Yaskawa INFORM job: PRINT3D17.JBI

/JOB
//NAME PRINT3D17
//POS
///NPOS 1138,0,0,0,0,0
///TOOL 9
///POSTYPE PULSE
///PULSE
C00000=35704,38341,-114719,81904,-122576,-81616,0
C00001=36579,38894,-113542,81280,-123389,-81453,0
C00002=42306,33068,-126081,74064,-124973,-85245,0
C00003=39937,31598,-129154,75978,-122913,-85572,0
C00004=34331,37524,-116454,82912,-121332,-81854,0
C00005=35234,38054,-115328,82245,-122145,-81700,0
C00006=34998,38355,-114678,82543,-122072,-81515,0
C00007=35467,38641,-114070,82205,-122503,-81430,0
C00008=35650,38409,-114572,81972,-122560,-81574,0
C00009=36212,38011,-115436,81348,-122827,-81855,0
C00010=36176,37331,-116893,81182,-122572,-82197,0
C00011=40262,33094,-125995,76081,-123713,-84903,0
C00012=40263,33039,-125991,76100,-123740,-84872,0
C00013=36399,37887,-115595,81173,-122955,-81890,0
C00014=41075,33073,-125931,75315,-124263,-84984,0
C00015=40068,32450,-127233,76121,-123383,-85125,0
C00016=35435,37299,-116842,81880,-122077,-82058,0
C00017=36321,37838,-115698,81229,-122883,-81904,0
C00018=35705,38292,-114715,81920,-122594,-81587,0
C00019=36579,38845,-113538,81297,-123409,-81425,0
C00020=42306,33013,-126077,74083,-125002,-85213,0
C00021=39937,31541,-129150,75996,-122940,-85539,0
C00022=34332,37475,-116451,82927,-121351,-81824,0
C00023=35234,38005,-115325,82261,-122164,-81671,0
C00024=34998,38306,-114675,82559,-122092,-81485,0
C00025=35467,38592,-114066,82221,-122522,-81401,0
C00026=35650,38360,-114568,81989,-122578,-81545,0
C00027=36212,37961,-115433,81364,-122847,-81826,0
C00028=36177,37281,-116890,81199,-122593,-82168,0
C00029=40263,33039,-125991,76100,-123740,-84872,0
C00030=40263,32984,-125988,76119,-123766,-84840,0
C00031=36400,37838,-115591,81189,-122975,-81861,0
C00032=41075,33018,-125927,75334,-124289,-84952,0
C00033=40068,32394,-127230,76140,-123410,-85093,0
C00034=35436,37249,-116838,81896,-122097,-82028,0
C00035=36322,37789,-115695,81246,-122903,-81874,0
C00036=35705,38243,-114712,81937,-122614,-81558,0
C00037=36579,38797,-113534,81314,-123427,-81396,0
C00038=42306,32958,-126074,74103,-125029,-85181,0
C00039=39938,31484,-129146,76015,-122968,-85507,0
C00040=34332,37425,-116447,82943,-121369,-81794,0
C00041=35235,37956,-115321,82277,-122183,-81642,0
C00042=34998,38257,-114671,82575,-122110,-81456,0
C00043=35467,38544,-114062,82237,-122540,-81372,0
C00044=35651,38311,-114564,82005,-122597,-81516,0
C00045=36213,37912,-115428,81381,-122867,-81797,0
C00046=36177,37232,-116886,81215,-122613,-82137,0
C00047=40263,32984,-125988,76119,-123766,-84840,0
C00048=40264,32929,-125983,76137,-123793,-84808,0
C00049=36400,37788,-115587,81206,-122994,-81831,0
C00050=41076,32964,-125923,75353,-124317,-84920,0
C00051=40069,32339,-127226,76159,-123437,-85061,0
C00052=35436,37199,-116833,81912,-122116,-81998,0
C00053=36322,37739,-115690,81263,-122923,-81845,0
C00054=35705,38194,-114708,81953,-122633,-81529,0
C00055=36580,38748,-113531,81331,-123447,-81367,0
C00056=42307,32903,-126069,74123,-125058,-85150,0
C00057=39938,31428,-129142,76033,-122995,-85474,0
C00058=34332,37375,-116443,82958,-121388,-81765,0
C00059=35235,37907,-115318,82293,-122201,-81612,0
C00060=34999,38208,-114667,82591,-122129,-81427,0
C00061=35468,38495,-114059,82254,-122560,-81343,0
C00062=35651,38262,-114561,82021,-122616,-81487,0
C00063=36213,37863,-115425,81398,-122886,-81767,0
C00064=36178,37182,-116883,81232,-122633,-82108,0
C00065=40264,32929,-125983,76137,-123793,-84808,0
C00066=40264,32874,-125980,76156,-123820,-84777,0
C00067=36400,37739,-115583,81223,-123015,-81802,0
C00068=41076,32909,-125919,75372,-124344,-84888,0
C00069=40069,32283,-127222,76177,-123463,-85029,0
C00070=35436,37150,-116830,81928,-122135,-81968,0
C00071=36322,37690,-115687,81279,-122942,-81816,0
C00072=35706,38145,-114704,81969,-122652,-81500,0
C00073=36580,38700,-113527,81348,-123466,-81338,0
C00074=42307,32849,-126066,74142,-125087,-85119,0
C00075=39938,31371,-129138,76052,-123023,-85442,0
C00076=34333,37326,-116439,82974,-121406,-81735,0
C00077=35235,37857,-115313,82310,-122221,-81583,0
C00078=34999,38160,-114663,82607,-122147,-81397,0
C00079=35468,38447,-114055,82270,-122578,-81314,0
C00080=35651,38214,-114557,82038,-122634,-81457,0
C00081=36213,37814,-115421,81414,-122906,-81738,0
C00082=36178,37132,-116878,81249,-122653,-82078,0
C00083=40264,32874,-125980,76156,-123820,-84777,0
C00084=40264,32820,-125975,76175,-123847,-84745,0
C00085=36401,37690,-115580,81240,-123034,-81772,0
C00086=41077,32854,-125915,75391,-124371,-84857,0
C00087=40070,32228,-127218,76196,-123491,-84997,0
C00088=35437,37100,-116827,81945,-122154,-81939,0
C00089=36323,37641,-115683,81296,-122962,-81786,0
C00090=35706,38096,-114700,81986,-122671,-81470,0
C00091=36580,38652,-113523,81365,-123486,-81309,0
C00092=42308,32794,-126061,74162,-125115,-85087,0
C00093=39939,31314,-129134,76070,-123050,-85409,0
C00094=34333,37276,-116436,82989,-121424,-81706,0
C00095=35236,37808,-115310,82326,-122239,-81554,0
C00096=34999,38111,-114660,82623,-122166,-81368,0
C00097=35468,38398,-114051,82286,-122597,-81284,0
C00098=35652,38165,-114553,82054,-122654,-81428,0
C00099=36214,37764,-115417,81431,-122925,-81709,0
C00100=36178,37082,-116875,81265,-122672,-82049,0
C00101=40264,32820,-125975,76175,-123847,-84745,0
C00102=40265,32765,-125972,76194,-123873,-84713,0
C00103=36401,37640,-115575,81256,-123054,-81743,0
C00104=41077,32800,-125911,75411,-124398,-84825,0
C00105=40070,32173,-127214,76215,-123517,-84965,0
C00106=35437,37050,-116822,81961,-122174,-81909,0
C00107=36323,37592,-115679,81313,-122981,-81757,0
C00108=35706,38048,-114696,82002,-122690,-81441,0
C00109=36580,38604,-113519,81382,-123505,-81280,0
C00110=42308,32739,-126058,74182,-125143,-85055,0
C00111=39939,31258,-129129,76089,-123078,-85376,0
C00112=34333,37226,-116431,83005,-121444,-81676,0
C00113=35236,37759,-115306,82342,-122259,-81524,0
C00114=35000,38062,-114656,82639,-122184,-81339,0
C00115=35469,38350,-114047,82303,-122615,-81255,0
C00116=35652,38116,-114549,82071,-122672,-81399,0
C00117=36214,37715,-115413,81448,-122946,-81679,0
C00118=36179,37032,-116870,81282,-122693,-82018,0
C00119=40265,32765,-125972,76194,-123873,-84713,0
C00120=40265,32711,-125967,76213,-123900,-84682,0
C00121=36401,37591,-115572,81273,-123073,-81713,0
C00122=41077,32745,-125906,75430,-124426,-84794,0
C00123=40070,32117,-127209,76233,-123545,-84933,0
C00124=35437,37000,-116819,81977,-122193,-81879,0
C00125=36323,37542,-115675,81330,-123002,-81727,0
C00126=35707,37999,-114692,82019,-122709,-81411,0
C00127=36581,38555,-113515,81399,-123525,-81251,0
C00128=42309,32685,-126053,74202,-125172,-85024,0
C00129=39940,31201,-129125,76108,-123106,-85344,0
C00130=34333,37177,-116427,83021,-121462,-81646,0
C00131=35236,37710,-115302,82358,-122277,-81494,0
C00132=35000,38013,-114651,82655,-122202,-81310,0
C00133=35469,38301,-114043,82319,-122634,-81226,0
C00134=35652,38067,-114545,82087,-122692,-81370,0
C00135=36214,37666,-115409,81465,-122965,-81649,0
C00136=36179,36982,-116867,81299,-122713,-81989,0
C00137=40265,32711,-125967,76213,-123900,-84682,0
C00138=40266,32656,-125962,76232,-123926,-84650,0
C00139=36402,37542,-115567,81290,-123094,-81684,0
C00140=41078,32691,-125903,75449,-124454,-84762,0
C00141=40071,32062,-127205,76252,-123571,-84901,0
C00142=35438,36951,-116814,81994,-122213,-81849,0
C00143=36324,37493,-115671,81347,-123022,-81697,0
C00144=35707,37950,-114688,82035,-122728,-81382,0
C00145=36581,38507,-113511,81416,-123545,-81222,0
C00146=42309,32630,-126049,74222,-125200,-84993,0
C00147=39940,31145,-129120,76126,-123133,-85311,0
C00148=34334,37127,-116423,83036,-121481,-81616,0
C00149=35237,37661,-115297,82374,-122295,-81465,0
C00150=35000,37965,-114647,82671,-122221,-81280,0
C00151=35469,38253,-114039,82335,-122653,-81197,0
C00152=35653,38019,-114541,82104,-122710,-81340,0
C00153=36215,37617,-115405,81481,-122985,-81620,0
C00154=36179,36933,-116862,81315,-122733,-81959,0
C00155=40266,32656,-125962,76232,-123926,-84650,0
C00156=40266,32601,-125958,76250,-123953,-84618,0
C00157=36402,37493,-115563,81307,-123114,-81655,0
C00158=41078,32636,-125898,75469,-124480,-84731,0
C00159=40071,32007,-127201,76271,-123597,-84869,0
C00160=35438,36901,-116809,82010,-122232,-81819,0
C00161=36324,37444,-115666,81363,-123041,-81668,0
C00162=35707,37901,-114684,82052,-122747,-81353,0
C00163=36581,38459,-113507,81433,-123563,-81193,0
C00164=42309,32575,-126044,74242,-125229,-84961,0
C00165=39940,31088,-129117,76145,-123161,-85278,0
C00166=34334,37078,-116419,83052,-121499,-81587,0
C00167=35237,37612,-115294,82391,-122315,-81435,0
C00168=35001,37916,-114643,82687,-122239,-81251,0
C00169=35470,38204,-114035,82352,-122671,-81168,0
C00170=35653,37970,-114537,82120,-122730,-81311,0
C00171=36215,37568,-115400,81498,-123004,-81591,0
C00172=36179,36883,-116859,81332,-122753,-81929,0
C00173=40266,32601,-125958,76250,-123953,-84618,0
C00174=40266,32547,-125953,76269,-123979,-84586,0
C00175=36402,37444,-115559,81324,-123133,-81625,0
C00176=41079,32582,-125893,75488,-124508,-84699,0
C00177=40072,31951,-127197,76290,-123625,-84836,0
C00178=35438,36851,-116805,82026,-122252,-81789,0
C00179=36324,37395,-115663,81380,-123061,-81638,0
C00180=35707,37853,-114679,82068,-122765,-81324,0
C00181=36582,38411,-113502,81450,-123582,-81163,0
C00182=42310,32521,-126039,74262,-125257,-84930,0
C00183=39941,31032,-129112,76164,-123188,-85245,0
C00184=34335,37028,-116414,83068,-121517,-81556,0
C00185=35237,37563,-115289,82407,-122333,-81406,0
C00186=35001,37867,-114639,82704,-122258,-81222,0
C00187=35470,38156,-114030,82368,-122690,-81139,0
C00188=35653,37921,-114532,82137,-122748,-81281,0
C00189=36215,37519,-115396,81515,-123024,-81561,0
C00190=36180,36833,-116854,81349,-122772,-81899,0
C00191=40266,32547,-125953,76269,-123979,-84586,0
C00192=40267,32493,-125949,76288,-124005,-84554,0
C00193=36403,37395,-115554,81341,-123153,-81595,0
C00194=41079,32527,-125889,75508,-124535,-84667,0
C00195=40072,31896,-127192,76309,-123651,-84804,0
C00196=35439,36802,-116801,82043,-122271,-81760,0
C00197=36325,37346,-115658,81397,-123080,-81609,0
C00198=35708,37804,-114675,82085,-122785,-81294,0
C00199=36582,38363,-113498,81467,-123602,-81134,0
C00200=42310,32466,-126035,74282,-125286,-84898,0
C00201=39941,30975,-129108,76183,-123216,-85213,0
C00202=34335,36979,-116411,83084,-121536,-81527,0
C00203=35237,37515,-115284,82423,-122353,-81376,0
C00204=35001,37819,-114634,82720,-122276,-81192,0
C00205=35470,38108,-114026,82385,-122708,-81109,0
C00206=35654,37873,-114528,82153,-122768,-81252,0
C00207=36216,37470,-115392,81532,-123044,-81532,0
C00208=36180,36784,-116850,81366,-122793,-81869,0
C00209=40267,32493,-125949,76288,-124005,-84554,0
C00210=40267,32438,-125944,76307,-124033,-84522,0
C00211=36403,37346,-115550,81358,-123172,-81566,0
C00212=41079,32473,-125884,75527,-124563,-84635,0
C00213=40072,31841,-127187,76328,-123679,-84772,0
C00214=35439,36752,-116797,82059,-122291,-81729,0
C00215=36325,37297,-115653,81414,-123101,-81579,0
C00216=35708,37756,-114671,82102,-122803,-81265,0
C00217=36583,38315,-113493,81484,-123622,-81105,0
C00218=42311,32412,-126030,74302,-125314,-84866,0
C00219=39942,30919,-129102,76202,-123243,-85180,0
C00220=34335,36930,-116406,83099,-121554,-81497,0
C00221=35238,37466,-115280,82440,-122371,-81346,0
C00222=35002,37770,-114630,82736,-122294,-81162,0
C00223=35471,38059,-114022,82401,-122728,-81080,0
C00224=35654,37825,-114523,82170,-122786,-81223,0
C00225=36216,37421,-115388,81549,-123063,-81502,0
C00226=36180,36734,-116845,81383,-122813,-81840,0
C00227=40267,32438,-125944,76307,-124033,-84522,0
C00228=40268,32384,-125939,76327,-124059,-84490,0
C00229=36403,37297,-115545,81375,-123193,-81536,0
C00230=41080,32419,-125880,75547,-124589,-84603,0
C00231=40073,31786,-127182,76347,-123705,-84739,0
C00232=35439,36703,-116792,82076,-122309,-81700,0
C00233=36325,37248,-115649,81431,-123121,-81550,0
C00234=35709,37707,-114666,82118,-122823,-81235,0
C00235=36583,38267,-113489,81502,-123641,-81076,0
C00236=42311,32358,-126026,74322,-125342,-84834,0
C00237=39942,30863,-129097,76221,-123271,-85147,0
C00238=34335,36880,-116401,83115,-121573,-81467,0
C00239=35238,37417,-115275,82456,-122390,-81317,0
C00240=35002,37722,-114625,82752,-122313,-81133,0
C00241=35471,38011,-114017,82418,-122746,-81050,0
C00242=35654,37776,-114519,82187,-122806,-81193,0
C00243=36216,37373,-115383,81566,-123083,-81472,0
C00244=36181,36685,-116840,81400,-122833,-81809,0
C00245=40268,32384,-125939,76327,-124059,-84490,0
C00246=40268,32330,-125935,76346,-124086,-84458,0
C00247=36404,37248,-115541,81392,-123212,-81507,0
C00248=41080,32364,-125875,75566,-124617,-84572,0
C00249=40073,31731,-127177,76366,-123733,-84707,0
C00250=35440,36653,-116788,82092,-122329,-81670,0
C00251=36326,37199,-115644,81448,-123140,-81520,0
C00252=35709,37659,-114661,82135,-122841,-81206,0
C00253=36583,38219,-113484,81519,-123659,-81046,0
C00254=42312,32303,-126021,74342,-125371,-84802,0
C00255=39943,30806,-129093,76240,-123299,-85114,0
C00256=34336,36831,-116397,83131,-121591,-81437,0
C00257=35239,37368,-115271,82472,-122409,-81287,0
C00258=35002,37673,-114621,82769,-122331,-81103,0
C00259=35471,37963,-114012,82434,-122764,-81021,0
C00260=35655,37728,-114514,82203,-122824,-81164,0
C00261=36217,37324,-115379,81583,-123102,-81443,0
C00262=36181,36635,-116836,81417,-122853,-81780,0
C00263=40268,32330,-125935,76346,-124086,-84458,0
C00264=40268,32275,-125930,76365,-124112,-84426,0
C00265=36404,37200,-115536,81410,-123232,-81476,0
C00266=41081,32310,-125869,75586,-124644,-84540,0
C00267=40074,31676,-127172,76385,-123759,-84675,0
C00268=35440,36604,-116783,82109,-122348,-81639,0
C00269=36326,37150,-115640,81465,-123160,-81490,0
C00270=35709,37610,-114657,82152,-122861,-81176,0
C00271=36583,38171,-113480,81536,-123679,-81017,0
C00272=42312,32249,-126016,74362,-125399,-84771,0
C00273=39943,30750,-129087,76259,-123326,-85081,0
C00274=34336,36782,-116392,83147,-121609,-81407,0
C00275=35239,37319,-115266,82489,-122428,-81258,0
C00276=35003,37625,-114616,82785,-122349,-81074,0
C00277=35472,37915,-114008,82451,-122783,-80992,0
C00278=35655,37679,-114510,82220,-122844,-81135,0
C00279=36217,37275,-115374,81600,-123122,-81413,0
C00280=36182,36586,-116831,81434,-122872,-81750,0
C00281=40268,32275,-125930,76365,-124112,-84426,0
C00282=40269,32221,-125924,76384,-124139,-84395,0
C00283=36404,37151,-115532,81427,-123252,-81447,0
C00284=41081,32256,-125865,75605,-124672,-84508,0
C00285=40074,31621,-127167,76404,-123786,-84642,0
C00286=35440,36555,-116777,82125,-122368,-81610,0
C00287=36326,37101,-115635,81483,-123179,-81461,0
C00288=35710,37562,-114652,82168,-122880,-81147,0
C00289=36584,38123,-113475,81553,-123699,-80988,0
C00290=42312,32195,-126011,74383,-125428,-84739,0
C00291=39943,30694,-129082,76278,-123354,-85048,0
C00292=34336,36733,-116386,83163,-121628,-81377,0
C00293=35239,37271,-115261,82505,-122446,-81228,0
C00294=35003,37576,-114611,82801,-122369,-81045,0
C00295=35472,37867,-114003,82467,-122802,-80962,0
C00296=35655,37631,-114505,82237,-122862,-81105,0
C00297=36217,37226,-115368,81617,-123141,-81384,0
C00298=36182,36536,-116827,81451,-122893,-81720,0
C00299=40269,32221,-125924,76384,-124139,-84395,0
C00300=40269,32167,-125920,76404,-124165,-84363,0
C00301=36405,37102,-115526,81444,-123271,-81417,0
C00302=41082,32202,-125859,75625,-124698,-84476,0
C00303=40074,31566,-127162,76423,-123813,-84610,0
C00304=35441,36505,-116773,82142,-122387,-81580,0
C00305=36327,37053,-115629,81500,-123200,-81431,0
C00306=35710,37513,-114647,82185,-122899,-81117,0
C00307=36584,38075,-113470,81571,-123718,-80959,0
C00308=42313,32140,-126006,74403,-125456,-84707,0
C00309=39944,30638,-129078,76297,-123381,-85015,0
C00310=34337,36683,-116382,83179,-121646,-81347,0
C00311=35239,37222,-115257,82522,-122466,-81198,0
C00312=35003,37528,-114606,82818,-122387,-81015,0
C00313=35472,37819,-113998,82484,-122821,-80933,0
C00314=35656,37583,-114500,82253,-122882,-81075,0
C00315=36218,37178,-115364,81634,-123161,-81353,0
C00316=36182,36487,-116821,81468,-122913,-81690,0
C00317=40269,32167,-125920,76404,-124165,-84363,0
C00318=40270,32113,-125914,76423,-124192,-84331,0
C00319=36405,37053,-115521,81461,-123292,-81388,0
C00320=41082,32148,-125854,75645,-124726,-84444,0
C00321=40075,31511,-127156,76443,-123840,-84577,0
C00322=35441,36456,-116768,82159,-122407,-81550,0
C00323=36327,37004,-115625,81517,-123219,-81401,0
C00324=35710,37465,-114642,82202,-122918,-81088,0
C00325=36584,38027,-113465,81588,-123738,-80930,0
C00326=42313,32086,-126000,74423,-125484,-84675,0
C00327=39944,30582,-129072,76316,-123409,-84982,0
C00328=34337,36634,-116377,83195,-121665,-81317,0
C00329=35240,37174,-115251,82538,-122484,-81168,0
C00330=35004,37480,-114601,82834,-122406,-80985,0
C00331=35472,37771,-113993,82501,-122839,-80904,0
C00332=35656,37534,-114495,82270,-122900,-81046,0
C00333=36218,37129,-115359,81651,-123180,-81324,0
C00334=36183,36438,-116816,81485,-122933,-81660,0
C00335=40270,32113,-125914,76423,-124192,-84331,0
C00336=40270,32059,-125910,76442,-124218,-84298,0
C00337=36405,37005,-115517,81478,-123311,-81357,0
C00338=41082,32094,-125849,75665,-124753,-84412,0
C00339=40075,31456,-127152,76462,-123867,-84545,0
C00340=35441,36407,-116762,82175,-122426,-81519,0
C00341=36327,36955,-115620,81534,-123239,-81371,0
C00342=35710,37417,-114637,82219,-122937,-81058,0
C00343=36585,37980,-113460,81605,-123757,-80900,0
C00344=42314,32032,-125996,74444,-125513,-84643,0
C00345=39945,30526,-129066,76335,-123437,-84949,0
C00346=34337,36585,-116372,83211,-121683,-81287,0
C00347=35240,37125,-115247,82555,-122502,-81139,0
C00348=35004,37432,-114596,82850,-122424,-80956,0
C00349=35473,37723,-113988,82517,-122857,-80874,0
C00350=35656,37486,-114490,82287,-122918,-81016,0
C00351=36218,37080,-115353,81668,-123200,-81294,0
C00352=36183,36388,-116812,81502,-122953,-81630,0
C00353=40270,32059,-125910,76442,-124218,-84298,0
C00354=40271,32005,-125904,76462,-124244,-84266,0
C00355=36406,36956,-115511,81496,-123331,-81328,0
C00356=41083,32040,-125844,75684,-124780,-84380,0
C00357=40076,31402,-127146,76481,-123894,-84513,0
C00358=35442,36358,-116758,82192,-122446,-81489,0
C00359=36328,36906,-115614,81551,-123258,-81341,0
C00360=35711,37369,-114632,82236,-122956,-81028,0
C00361=36585,37932,-113455,81623,-123776,-80871,0
C00362=42314,31978,-125990,74464,-125542,-84612,0
C00363=39945,30470,-129061,76354,-123464,-84916,0
C00364=34338,36536,-116367,83227,-121701,-81257,0
C00365=35240,37077,-115241,82572,-122522,-81109,0
C00366=35004,37383,-114591,82867,-122443,-80926,0
C00367=35473,37675,-113983,82534,-122876,-80844,0
C00368=35657,37438,-114485,82304,-122938,-80987,0
C00369=36219,37032,-115349,81685,-123219,-81265,0
C00370=36183,36339,-116806,81519,-122972,-81599,0
C00371=40271,32005,-125904,76462,-124244,-84266,0
C00372=40271,31951,-125898,76481,-124272,-84234,0
C00373=36406,36908,-115506,81513,-123350,-81298,0
C00374=41083,31986,-125838,75704,-124807,-84348,0
C00375=40076,31347,-127140,76501,-123920,-84480,0
C00376=35442,36308,-116752,82209,-122464,-81459,0
C00377=36328,36858,-115610,81569,-123278,-81312,0
C00378=35711,37320,-114627,82253,-122975,-80999,0
C00379=36585,37884,-113450,81640,-123795,-80842,0
C00380=42315,31924,-125984,74485,-125569,-84580,0
C00381=39945,30414,-129056,76374,-123492,-84883,0
C00382=34338,36487,-116361,83243,-121720,-81227,0
C00383=35241,37028,-115236,82588,-122540,-81080,0
C00384=35005,37335,-114586,82883,-122461,-80896,0
C00385=35474,37627,-113978,82551,-122895,-80815,0
C00386=35657,37390,-114480,82321,-122956,-80957,0
C00387=36219,36983,-115343,81703,-123239,-81234,0
C00388=36184,36290,-116801,81536,-122993,-81569,0
C00389=40271,31951,-125898,76481,-124272,-84234,0
C00390=40271,31897,-125892,76501,-124298,-84202,0
C00391=36406,36859,-115500,81530,-123371,-81268,0
C00392=41084,31932,-125833,75724,-124835,-84316,0
C00393=40076,31292,-127135,76520,-123948,-84447,0
C00394=35442,36259,-116747,82226,-122484,-81429,0
C00395=36328,36809,-115604,81586,-123297,-81281,0
C00396=35711,37272,-114621,82270,-122994,-80969,0
C00397=36586,37837,-113444,81658,-123815,-80812,0
C00398=42315,31870,-125978,74505,-125598,-84548,0
C00399=39946,30358,-129050,76393,-123519,-84849,0
C00400=34338,36438,-116357,83259,-121738,-81197,0
C00401=35241,36980,-115230,82605,-122560,-81049,0
C00402=35005,37287,-114581,82900,-122479,-80867,0
C00403=35474,37579,-113972,82568,-122914,-80785,0
C00404=35657,37342,-114474,82338,-122976,-80927,0
C00405=36219,36935,-115338,81720,-123258,-81205,0
C00406=36184,36241,-116796,81554,-123013,-81539,0
C00407=40271,31897,-125892,76501,-124298,-84202,0
C00408=40272,31843,-125888,76520,-124325,-84170,0
C00409=36407,36811,-115495,81548,-123391,-81238,0
C00410=41084,31878,-125827,75744,-124863,-84284,0
C00411=40077,31238,-127129,76539,-123974,-84415,0
C00412=35443,36210,-116742,82242,-122503,-81399,0
C00413=36329,36761,-115598,81603,-123318,-81252,0
C00414=35712,37224,-114616,82287,-123013,-80939,0
C00415=36586,37789,-113439,81675,-123834,-80783,0
C00416=42315,31816,-125973,74526,-125627,-84516,0
C00417=39946,30302,-129044,76412,-123547,-84816,0
C00418=34339,36389,-116351,83275,-121756,-81167,0
C00419=35241,36931,-115226,82622,-122578,-81020,0
C00420=35005,37239,-114575,82916,-122498,-80837,0
C00421=35474,37531,-113967,82585,-122932,-80756,0
C00422=35658,37294,-114469,82355,-122994,-80898,0
C00423=36220,36887,-115333,81737,-123278,-81175,0
C00424=36184,36192,-116790,81571,-123032,-81509,0
C00425=40272,31843,-125888,76520,-124325,-84170,0
C00426=40272,31789,-125882,76540,-124351,-84138,0
C00427=36407,36762,-115490,81565,-123410,-81208,0
C00428=41084,31824,-125821,75764,-124889,-84252,0
C00429=40077,31183,-127123,76559,-124001,-84382,0
C00430=35443,36161,-116736,82259,-122523,-81368,0
C00431=36329,36712,-115592,81621,-123338,-81222,0
C00432=35712,37176,-114611,82304,-123032,-80909,0
C00433=36586,37742,-113434,81693,-123854,-80753,0
C00434=42316,31762,-125968,74546,-125654,-84484,0
C00435=39947,30246,-129039,76432,-123574,-84783,0
C00436=34339,36341,-116345,83292,-121775,-81136,0
C00437=35242,36883,-115220,82638,-122597,-80990,0
C00438=35006,37191,-114570,82933,-122516,-80807,0
C00439=35474,37483,-113962,82601,-122950,-80726,0
C00440=35658,37246,-114463,82371,-123014,-80868,0
C00441=36220,36838,-115327,81754,-123297,-81145,0
C00442=36185,36143,-116784,81588,-123053,-81479,0
C00443=40272,31789,-125882,76540,-124351,-84138,0
C00444=40273,31735,-125876,76559,-124378,-84106,0
C00445=36407,36714,-115484,81583,-123430,-81179,0
C00446=41085,31770,-125815,75784,-124917,-84219,0
C00447=40078,31128,-127117,76578,-124028,-84350,0
C00448=35443,36112,-116730,82276,-122543,-81338,0
C00449=36329,36664,-115588,81638,-123357,-81192,0
C00450=35713,37128,-114605,82321,-123050,-80880,0
C00451=36587,37694,-113428,81710,-123872,-80724,0
C00452=42316,31708,-125961,74567,-125683,-84452,0
C00453=39947,30191,-129033,76451,-123602,-84750,0
C00454=34339,36292,-116339,83308,-121793,-81106,0
C00455=35242,36835,-115214,82655,-122616,-80960,0
C00456=35006,37143,-114564,82949,-122534,-80777,0
C00457=35475,37436,-113956,82618,-122969,-80697,0
C00458=35658,37198,-114458,82388,-123032,-80838,0
C00459=36220,36790,-115322,81772,-123317,-81115,0
C00460=36185,36094,-116779,81605,-123072,-81449,0
C00461=40273,31735,-125876,76559,-124378,-84106,0
C00462=40273,31682,-125869,76579,-124404,-84073,0
C00463=36408,36665,-115479,81600,-123449,-81149,0
C00464=41085,31717,-125810,75804,-124944,-84187,0
C00465=40078,31074,-127112,76598,-124055,-84317,0
C00466=35444,36063,-116724,82293,-122562,-81308,0
C00467=36330,36615,-115582,81655,-123377,-81162,0
C00468=35713,37080,-114599,82338,-123070,-80850,0
C00469=36587,37647,-113422,81728,-123892,-80694,0
C00470=42317,31655,-125955,74588,-125712,-84420,0
C00471=39948,30135,-129026,76471,-123630,-84717,0
C00472=34340,36243,-116334,83324,-121812,-81076,0
C00473=35242,36786,-115209,82672,-122634,-80930,0
C00474=35006,37095,-114559,82966,-122553,-80748,0
C00475=35475,37388,-113950,82635,-122988,-80667,0
C00476=35659,37150,-114452,82405,-123052,-80809,0
C00477=36221,36742,-115317,81789,-123337,-81085,0
C00478=36185,36045,-116774,81623,-123093,-81418,0
C00479=40273,31682,-125869,76579,-124404,-84073,0
C00480=40273,31628,-125864,76599,-124431,-84041,0
C00481=36408,36617,-115473,81618,-123469,-81118,0
C00482=41086,31663,-125804,75824,-124971,-84155,0
C00483=40079,31020,-127106,76617,-124082,-84285,0
C00484=35444,36014,-116719,82310,-122582,-81278,0
C00485=36330,36567,-115576,81673,-123396,-81132,0
C00486=35713,37032,-114594,82355,-123088,-80820,0
C00487=36587,37599,-113417,81746,-123911,-80665,0
C00488=42317,31601,-125950,74608,-125741,-84388,0
C00489=39948,30079,-129020,76490,-123657,-84684,0
C00490=34340,36194,-116328,83340,-121830,-81046,0
C00491=35243,36738,-115203,82689,-122653,-80900,0
C00492=35006,37047,-114553,82983,-122571,-80718,0
C00493=35475,37340,-113945,82652,-123007,-80637,0
C00494=35659,37102,-114447,82423,-123070,-80779,0
C00495=36221,36693,-115311,81807,-123356,-81055,0
C00496=36186,35996,-116768,81640,-123112,-81388,0
C00497=40273,31628,-125864,76599,-124431,-84041,0
C00498=40274,31574,-125858,76618,-124457,-84009,0
C00499=36408,36569,-115467,81635,-123489,-81089,0
C00500=41086,31609,-125798,75844,-124998,-84123,0
C00501=40079,30965,-127100,76637,-124109,-84252,0
C00502=35444,35965,-116713,82327,-122600,-81248,0
C00503=36330,36519,-115571,81690,-123416,-81102,0
C00504=35713,36984,-114588,82372,-123108,-80791,0
C00505=36588,37552,-113411,81763,-123931,-80635,0
C00506=42318,31547,-125944,74629,-125768,-84356,0
C00507=39948,30024,-129015,76510,-123684,-84650,0
C00508=35603,34554,-119651,81803,-122284,-81944,0
C00509=35599,34552,-119656,81806,-122280,-81945,0
C00510=35261,34964,-118796,82221,-122166,-81703,0
C00511=35265,34966,-118792,82218,-122168,-81703,0
C00512=34340,36146,-116322,83357,-121848,-81016,0
C00513=35243,36690,-115197,82705,-122672,-80870,0
C00514=35007,36999,-114547,82999,-122590,-80688,0
C00515=35476,37293,-113939,82669,-123025,-80608,0
C00516=35659,37054,-114441,82440,-123088,-80749,0
C00517=36221,36645,-115305,81824,-123376,-81026,0
C00518=36186,35947,-116762,81657,-123132,-81358,0
C00519=40274,31574,-125858,76618,-124457,-84009,0
C00520=40274,31521,-125852,76638,-124483,-83976,0
C00521=36409,36520,-115461,81653,-123509,-81059,0
C00522=41086,31556,-125791,75865,-125026,-84091,0
C00523=40079,30911,-127093,76657,-124135,-84219,0
C00524=35445,35917,-116707,82344,-122619,-81217,0
C00525=36331,36470,-115565,81708,-123437,-81072,0
C00526=35714,36937,-114582,82389,-123126,-80760,0
C00527=36588,37505,-113405,81781,-123950,-80605,0
C00528=42318,31493,-125938,74650,-125797,-84323,0
C00529=39949,29968,-129008,76530,-123711,-84617,0
C00530=35603,34504,-119645,81820,-122303,-81913,0
C00531=35585,34493,-119667,81834,-122287,-81916,0
C00532=35247,34905,-118808,82249,-122172,-81675,0
C00533=35265,34916,-118786,82235,-122189,-81672,0
C00534=34341,36097,-116316,83373,-121867,-80985,0
C00535=35243,36642,-115191,82722,-122691,-80840,0
C00536=35007,36951,-114541,83016,-122608,-80658,0
C00537=35476,37245,-113933,82686,-123044,-80578,0
C00538=35659,37007,-114435,82457,-123108,-80719,0
C00539=36222,36597,-115298,81841,-123395,-80995,0
C00540=36186,35898,-116755,81675,-123153,-81327,0
C00541=40274,31521,-125852,76638,-124483,-83976,0
C00542=40275,31467,-125845,76658,-124510,-83944,0
C00543=36409,36472,-115455,81670,-123528,-81028,0
C00544=41087,31502,-125785,75885,-125052,-84059,0
C00545=40080,30856,-127087,76676,-124163,-84186,0
C00546=35445,35868,-116701,82361,-122639,-81187,0
C00547=36331,36422,-115558,81726,-123456,-81042,0
C00548=35714,36889,-114576,82406,-123146,-80731,0
C00549=36588,37457,-113399,81799,-123969,-80576,0
C00550=42318,31440,-125931,74671,-125826,-84291,0
C00551=39949,29913,-129002,76549,-123739,-84584,0
C00552=35604,34453,-119640,81837,-122324,-81882,0
C00553=35571,34434,-119679,81862,-122295,-81887,0
C00554=35233,34847,-118819,82276,-122179,-81646,0
C00555=35266,34866,-118779,82252,-122208,-81641,0
C00556=34341,36048,-116311,83389,-121885,-80955,0
C00557=35244,36594,-115186,82739,-122709,-80810,0
C00558=35007,36904,-114535,83033,-122626,-80628,0
C00559=35476,37198,-113927,82703,-123062,-80548,0
C00560=35660,36959,-114429,82474,-123126,-80690,0
C00561=36222,36549,-115292,81859,-123415,-80965,0
C00562=36187,35849,-116750,81692,-123172,-81297,0
C00563=40275,31467,-125845,76658,-124510,-83944,0
C00564=40275,31413,-125839,76678,-124536,-83912,0
C00565=36409,36424,-115449,81688,-123548,-80999,0
C00566=41087,31449,-125779,75905,-125080,-84026,0
C00567=40080,30802,-127081,76696,-124189,-84154,0
C00568=35445,35819,-116696,82378,-122659,-81157,0
C00569=36331,36374,-115552,81743,-123476,-81012,0
C00570=35714,36841,-114570,82423,-123164,-80701,0
C00571=36589,37410,-113393,81816,-123988,-80546,0
C00572=42319,31386,-125926,74692,-125853,-84259,0
C00573=39950,29857,-128995,76569,-123766,-84551,0
C00574=35604,34403,-119633,81854,-122345,-81851,0
C00575=35557,34375,-119690,81890,-122302,-81858,0
C00576=35219,34789,-118831,82304,-122186,-81617,0
C00577=35266,34817,-118773,82269,-122228,-81610,0
C00578=34341,36000,-116305,83405,-121904,-80925,0
C00579=35244,36546,-115180,82756,-122729,-80780,0
C00580=35008,36856,-114529,83050,-122645,-80598,0
C00581=35477,37150,-113921,82720,-123081,-80518,0
C00582=35660,36911,-114423,82491,-123146,-80659,0
C00583=36222,36501,-115287,81876,-123434,-80936,0
C00584=36187,35801,-116744,81710,-123192,-81267,0
C00585=40275,31413,-125839,76678,-124536,-83912,0
C00586=40275,31360,-125833,76698,-124563,-83879,0
C00587=36410,36376,-115443,81706,-123568,-80969,0
C00588=41088,31395,-125773,75926,-125107,-83994,0
C00589=40081,30748,-127075,76716,-124216,-84121,0
C00590=35446,35770,-116689,82395,-122678,-81126,0
C00591=36332,36326,-115546,81761,-123495,-80981,0
C00592=35715,36793,-114564,82441,-123184,-80671,0
C00593=36589,37363,-113387,81834,-124008,-80517,0
C00594=42319,31333,-125919,74713,-125882,-84227,0
C00595=39950,29802,-128988,76589,-123794,-84517,0
C00596=35604,34353,-119627,81872,-122364,-81819,0
C00597=35543,34317,-119702,81918,-122309,-81829,0
C00598=35205,34730,-118842,82332,-122192,-81588,0
C00599=35266,34767,-118768,82286,-122247,-81579,0
C00600=34342,35951,-116298,83422,-121922,-80894,0
C00601=35244,36498,-115173,82773,-122747,-80750,0
C00602=35008,36808,-114523,83066,-122663,-80568,0
C00603=35477,37103,-113915,82737,-123100,-80489,0
C00604=35660,36863,-114417,82508,-123164,-80630,0
C00605=36223,36453,-115281,81894,-123454,-80905,0
C00606=36187,35752,-116738,81727,-123212,-81237,0
C00607=40275,31360,-125833,76698,-124563,-83879,0
C00608=40276,31307,-125827,76718,-124590,-83847,0
C00609=36410,36328,-115436,81723,-123588,-80938,0
C00610=41088,31342,-125766,75946,-125134,-83962,0
C00611=40081,30694,-127068,76736,-124243,-84088,0
C00612=35446,35722,-116683,82412,-122698,-81096,0
C00613=36332,36278,-115540,81778,-123515,-80951,0
C00614=35715,36746,-114558,82458,-123202,-80641,0
C00615=36589,37316,-113381,81852,-124027,-80487,0
C00616=42320,31279,-125912,74734,-125911,-84194,0
C00617=39951,29746,-128982,76608,-123822,-84484,0
C00618=35605,34303,-119620,81889,-122385,-81789,0
C00619=35528,34258,-119713,81946,-122317,-81800,0
C00620=35190,34672,-118853,82360,-122199,-81559,0
C00621=35267,34717,-118761,82303,-122268,-81548,0
C00622=34342,35903,-116292,83438,-121940,-80864,0
C00623=35245,36450,-115167,82790,-122765,-80720,0
C00624=35008,36761,-114517,83083,-122682,-80539,0
C00625=35477,37055,-113909,82754,-123118,-80459,0
C00626=35661,36816,-114411,82526,-123184,-80600,0
C00627=36223,36405,-115274,81912,-123473,-80875,0
C00628=36188,35703,-116731,81745,-123232,-81206,0
C00629=40276,31307,-125827,76718,-124590,-83847,0
C00630=40276,31253,-125820,76738,-124617,-83814,0
C00631=36410,36280,-115430,81741,-123608,-80908,0
C00632=41089,31289,-125759,75966,-125161,-83929,0
C00633=40082,30640,-127061,76756,-124270,-84055,0
C00634=35446,35673,-116676,82429,-122716,-81065,0
C00635=36332,36230,-115534,81796,-123534,-80922,0
C00636=35715,36698,-114551,82475,-123222,-80611,0
C00637=36590,37268,-113375,81870,-124046,-80457,0
C00638=42320,31226,-125906,74755,-125938,-84162,0
C00639=39951,29691,-128975,76628,-123849,-84450,0
C00640=35605,34253,-119614,81906,-122406,-81757,0
C00641=35514,34199,-119724,81974,-122324,-81771,0
C00642=35176,34614,-118864,82387,-122206,-81530,0
C00643=35267,34668,-118755,82320,-122287,-81518,0
C00644=34342,35854,-116285,83455,-121959,-80833,0
C00645=35245,36402,-115160,82807,-122785,-80690,0
C00646=35009,36713,-114511,83100,-122700,-80509,0
C00647=35478,37008,-113902,82772,-123137,-80429,0
C00648=35661,36768,-114404,82543,-123202,-80570,0
C00649=36223,36357,-115268,81929,-123493,-80845,0
C00650=36188,35655,-116725,81763,-123252,-81176,0
C00651=40276,31253,-125820,76738,-124617,-83814,0
C00652=40277,31200,-125813,76758,-124643,-83782,0
C00653=36411,36232,-115423,81759,-123627,-80878,0
C00654=41089,31235,-125753,75987,-125189,-83897,0
C00655=40082,30586,-127054,76776,-124296,-84023,0
C00656=35447,35625,-116670,82446,-122736,-81035,0
C00657=36333,36182,-115527,81814,-123554,-80891,0
C00658=35716,36650,-114545,82492,-123240,-80581,0
C00659=36590,37221,-113368,81888,-124065,-80428,0
C00660=42320,31172,-125899,74776,-125967,-84130,0
C00661=39951,29636,-128969,76648,-123877,-84417,0
C00662=35606,34203,-119608,81923,-122425,-81726,0
C00663=35500,34141,-119735,82002,-122331,-81741,0
C00664=35162,34556,-118876,82415,-122213,-81502,0
C00665=35267,34618,-118748,82337,-122307,-81486,0
C00666=34343,35806,-116280,83471,-121977,-80803,0
C00667=35245,36354,-115155,82824,-122803,-80659,0
C00668=35009,36665,-114504,83117,-122718,-80478,0
C00669=35478,36961,-113896,82789,-123155,-80399,0
C00670=35662,36721,-114398,82560,-123221,-80540,0
C00671=36224,36309,-115261,81947,-123512,-80815,0
C00672=36188,35606,-116719,81780,-123272,-81145,0
C00673=40277,31200,-125813,76758,-124643,-83782,0
C00674=40277,31146,-125806,76778,-124670,-83749,0
C00675=36411,36184,-115418,81776,-123647,-80848,0
C00676=41089,31182,-125746,76007,-125215,-83864,0
C00677=40082,30531,-127048,76796,-124324,-83990,0
C00678=35447,35576,-116663,82464,-122755,-81004,0
C00679=36333,36134,-115521,81831,-123574,-80861,0
C00680=35716,36603,-114539,82510,-123260,-80551,0
C00681=36590,37174,-113362,81905,-124085,-80398,0
C00682=42321,31119,-125892,74797,-125996,-84098,0
C00683=39952,29581,-128962,76668,-123904,-84384,0
C00684=35606,34153,-119601,81941,-122446,-81695,0
C00685=35486,34082,-119745,82030,-122339,-81712,0
C00686=35148,34498,-118886,82443,-122220,-81473,0
C00687=35268,34568,-118741,82354,-122326,-81456,0
C00688=34343,35758,-116273,83488,-121996,-80773,0
C00689=35246,36306,-115148,82841,-122822,-80629,0
C00690=35009,36618,-114498,83134,-122737,-80449,0
C00691=35478,36913,-113890,82806,-123173,-80369,0
C00692=35662,36673,-114392,82577,-123240,-80510,0
C00693=36224,36261,-115256,81964,-123532,-80785,0
C00694=36189,35557,-116712,81798,-123292,-81115,0
C00695=40277,31146,-125806,76778,-124670,-83749,0
C00696=40277,31093,-125799,76798,-124696,-83717,0
C00697=36411,36136,-115411,81794,-123666,-80818,0
C00698=41090,31129,-125739,76028,-125243,-83832,0
C00699=40083,30478,-127041,76816,-124350,-83956,0
C00700=35447,35528,-116657,82481,-122775,-80974,0
C00701=36333,36086,-115514,81849,-123594,-80831,0
C00702=35716,36555,-114532,82527,-123278,-80521,0
C00703=36591,37127,-113355,81923,-124104,-80369,0
C00704=42321,31066,-125885,74818,-126023,-84066,0
C00705=39952,29525,-128955,76688,-123932,-84350,0
C00706=35606,34103,-119595,81958,-122467,-81664,0
C00707=35471,34023,-119757,82059,-122346,-81683,0
C00708=35134,34440,-118896,82471,-122226,-81444,0
C00709=35268,34519,-118735,82371,-122347,-81425,0
C00710=34343,35709,-116267,83504,-122014,-80742,0
C00711=35246,36259,-115142,82858,-122840,-80599,0
C00712=35010,36570,-114491,83151,-122755,-80419,0
C00713=35479,36866,-113883,82823,-123193,-80340,0
C00714=35662,36626,-114385,82595,-123258,-80480,0
C00715=36224,36213,-115249,81982,-123551,-80755,0
C00716=36189,35509,-116706,81816,-123311,-81084,0
C00717=40277,31093,-125799,76798,-124696,-83717,0
C00718=40278,31040,-125792,76818,-124722,-83684,0
C00719=36412,36088,-115404,81812,-123686,-80788,0
C00720=41090,31076,-125733,76048,-125271,-83800,0
C00721=40083,30424,-127035,76836,-124377,-83924,0
C00722=35448,35479,-116651,82498,-122794,-80943,0
C00723=36334,36038,-115507,81867,-123614,-80800,0
C00724=35717,36508,-114525,82545,-123297,-80491,0
C00725=36591,37080,-113349,81941,-124124,-80339,0
C00726=42322,31012,-125878,74840,-126052,-84033,0
C00727=39953,29470,-128948,76708,-123959,-84316,0
C00728=35607,34053,-119588,81975,-122486,-81632,0
C00729=35457,33965,-119767,82087,-122353,-81653,0
C00730=35119,34381,-118908,82499,-122233,-81415,0
C00731=35268,34470,-118728,82388,-122367,-81393,0
C00732=34344,35661,-116260,83521,-122032,-80712,0
C00733=35246,36211,-115135,82875,-122860,-80569,0
C00734=35010,36523,-114485,83168,-122773,-80388,0
C00735=35479,36819,-113877,82840,-123211,-80309,0
C00736=35662,36578,-114378,82612,-123278,-80450,0
C00737=36225,36165,-115242,82000,-123571,-80724,0
C00738=36189,35461,-116699,81833,-123332,-81054,0
C00739=40278,31040,-125792,76818,-124722,-83684,0
C00740=40278,30987,-125785,76838,-124749,-83652,0
C00741=36412,36040,-115397,81830,-123705,-80757,0
C00742=41091,31022,-125726,76069,-125297,-83767,0
C00743=40084,30370,-127027,76856,-124404,-83891,0
C00744=35448,35431,-116644,82515,-122813,-80913,0
C00745=36334,35990,-115500,81885,-123633,-80770,0
C00746=35717,36460,-114519,82562,-123316,-80461,0
C00747=36591,37034,-113342,81959,-124142,-80309,0
C00748=42322,30959,-125872,74861,-126081,-84001,0
C00749=39953,29415,-128941,76728,-123987,-84283,0
C00750=35607,34004,-119581,81993,-122507,-81601,0
C00751=35443,33906,-119779,82115,-122361,-81624,0
C00752=35105,34323,-118918,82526,-122240,-81386,0
C00753=35269,34420,-118722,82405,-122386,-81363,0
C00754=34344,35613,-116253,83537,-122051,-80681,0
C00755=35247,36163,-115128,82892,-122878,-80539,0
C00756=35010,36475,-114478,83185,-122792,-80358,0
C00757=35479,36772,-113870,82858,-123230,-80280,0
C00758=35663,36531,-114372,82630,-123296,-80420,0
C00759=36225,36118,-115235,82018,-123591,-80694,0
C00760=36190,35412,-116692,81851,-123352,-81023,0
C00761=40278,30987,-125785,76838,-124749,-83652,0
C00762=40279,30934,-125779,76858,-124775,-83619,0
C00763=36412,35993,-115391,81848,-123726,-80727,0
C00764=41091,30969,-125719,76090,-125325,-83735,0
C00765=40084,30316,-127020,76876,-124431,-83858,0
C00766=35448,35382,-116637,82533,-122832,-80882,0
C00767=36334,35942,-115495,81903,-123653,-80740,0
C00768=35717,36413,-114512,82580,-123335,-80431,0
C00769=36592,36987,-113335,81977,-124162,-80279,0
C00770=42323,30906,-125865,74882,-126108,-83968,0
C00771=39953,29360,-128933,76748,-124015,-84249,0
C00772=35607,33954,-119574,82010,-122528,-81570,0
C00773=35429,33848,-119789,82143,-122368,-81595,0
C00774=35091,34265,-118928,82554,-122246,-81357,0
C00775=35269,34371,-118715,82423,-122406,-81331,0
C00776=34344,35565,-116246,83554,-122069,-80651,0
C00777=35247,36115,-115121,82910,-122896,-80509,0
C00778=35011,36428,-114471,83202,-122810,-80329,0
C00779=35480,36725,-113863,82875,-123248,-80250,0
C00780=35663,36484,-114365,82647,-123315,-80390,0
C00781=36225,36070,-115228,82035,-123610,-80664,0
C00782=36190,35364,-116685,81869,-123371,-80992,0
C00783=40279,30934,-125779,76858,-124775,-83619,0
C00784=40279,30881,-125772,76878,-124802,-83586,0
C00785=36413,35945,-115384,81866,-123746,-80697,0
C00786=41091,30916,-125711,76110,-125352,-83702,0
C00787=40084,30262,-127013,76896,-124457,-83825,0
C00788=35449,35334,-116630,82550,-122852,-80851,0
C00789=36335,35894,-115488,81921,-123672,-80710,0
C00790=35718,36366,-114505,82597,-123354,-80401,0
C00791=36592,36940,-113328,81995,-124181,-80249,0
C00792=42323,30853,-125858,74903,-126137,-83936,0
C00793=39954,29305,-128926,76768,-124042,-84216,0
C00794=35608,33904,-119567,82028,-122547,-81538,0
C00795=35425,33795,-119787,82164,-122384,-81564,0
C00796=35087,34213,-118927,82575,-122262,-81326,0
C00797=35269,34322,-118708,82440,-122425,-81300,0
C00798=34344,35517,-116239,83571,-122087,-80620,0
C00799=35247,36068,-115114,82927,-122916,-80478,0
C00800=35011,36381,-114465,83219,-122829,-80298,0
C00801=35480,36678,-113856,82892,-123266,-80220,0
C00802=35663,36436,-114358,82665,-123334,-80359,0
C00803=36226,36022,-115221,82053,-123630,-80634,0
C00804=36190,35315,-116678,81887,-123392,-80962,0
C00805=40279,30881,-125772,76878,-124802,-83586,0
C00806=40279,30828,-125764,76899,-124828,-83554,0
C00807=36413,35897,-115378,81884,-123765,-80666,0
C00808=41092,30863,-125704,76131,-125379,-83669,0
C00809=40085,30208,-127006,76916,-124485,-83792,0
C00810=35449,35286,-116623,82567,-122871,-80821,0
C00811=36335,35847,-115480,81938,-123692,-80679,0
C00812=35718,36318,-114498,82615,-123372,-80370,0
C00813=36592,36893,-113322,82014,-124201,-80220,0
C00814=42323,30800,-125850,74925,-126166,-83903,0
C00815=39954,29250,-128919,76788,-124069,-84182,0
C00816=35608,33854,-119560,82045,-122568,-81507,0
C00817=35425,33746,-119780,82181,-122405,-81533,0
C00818=35087,34164,-118919,82592,-122282,-81295,0
C00819=35270,34272,-118701,82457,-122446,-81269,0
C00820=34345,35469,-116232,83587,-122106,-80590,0
C00821=35248,36020,-115107,82944,-122934,-80448,0
C00822=35011,36334,-114458,83236,-122847,-80268,0
C00823=35480,36631,-113849,82910,-123285,-80190,0
C00824=35664,36389,-114351,82682,-123353,-80330,0
C00825=36226,35975,-115214,82071,-123649,-80604,0
C00826=36191,35267,-116671,81904,-123411,-80932,0
C00827=40279,30828,-125764,76899,-124828,-83554,0
C00828=40280,30775,-125757,76919,-124855,-83521,0
C00829=36413,35850,-115369,81902,-123785,-80636,0
C00830=41092,30811,-125697,76152,-125406,-83637,0
C00831=40085,30155,-126998,76936,-124511,-83759,0
C00832=35449,35238,-116616,82585,-122891,-80791,0
C00833=36335,35799,-115473,81957,-123711,-80649,0
C00834=35718,36271,-114491,82632,-123392,-80340,0
C00835=36593,36846,-113315,82032,-124219,-80189,0
C00836=42324,30747,-125843,74946,-126193,-83871,0
C00837=39955,29195,-128911,76809,-124096,-84149,0
C00838=35608,33805,-119552,82063,-122588,-81476,0
C00839=35425,33696,-119773,82199,-122424,-81501,0
C00840=35088,34115,-118912,82609,-122301,-81264,0
C00841=35270,34223,-118694,82475,-122466,-81238,0
C00842=34345,35421,-116226,83604,-122124,-80559,0
C00843=35248,35973,-115101,82961,-122953,-80418,0
C00844=35012,36286,-114451,83253,-122865,-80238,0
C00845=35481,36584,-113842,82927,-123303,-80160,0
C00846=35664,36342,-114344,82699,-123371,-80300,0
C00847=36226,35927,-115207,82089,-123669,-80574,0
C00848=36191,35219,-116665,81922,-123431,-80901,0
C00849=40280,30775,-125757,76919,-124855,-83521,0
C00850=40280,30722,-125750,76939,-124881,-83488,0
C00851=36414,35802,-115363,81920,-123804,-80606,0
C00852=41093,30758,-125689,76173,-125433,-83604,0
C00853=40086,30101,-126991,76957,-124537,-83726,0
C00854=35450,35189,-116608,82602,-122909,-80760,0
C00855=36336,35751,-115466,81974,-123731,-80619,0
C00856=35719,36224,-114484,82650,-123410,-80310,0
C00857=36593,36800,-113308,82050,-124239,-80160,0
C00858=42324,30694,-125835,74968,-126222,-83838,0
C00859=39955,29141,-128904,76829,-124124,-84115,0
C00860=35609,33755,-119546,82080,-122608,-81444,0
C00861=35426,33646,-119765,82216,-122445,-81470,0
C00862=35088,34066,-118905,82626,-122322,-81233,0
C00863=35270,34174,-118686,82492,-122485,-81207,0
C00864=34345,35373,-116219,83621,-122143,-80528,0
C00865=35248,35925,-115094,82979,-122971,-80387,0
C00866=35012,36239,-114443,83270,-122884,-80208,0
C00867=35481,36537,-113835,82945,-123323,-80130,0
C00868=35664,36295,-114337,82717,-123391,-80269,0
C00869=36227,35879,-115201,82107,-123688,-80543,0
C00870=36191,35171,-116658,81940,-123451,-80870,0
C00871=40280,30722,-125750,76939,-124881,-83488,0
C00872=40281,30669,-125742,76960,-124907,-83456,0
C00873=36414,35754,-115356,81938,-123824,-80575,0
C00874=41093,30705,-125682,76193,-125460,-83572,0
C00875=40086,30047,-126983,76977,-124564,-83692,0
C00876=35450,35141,-116601,82620,-122929,-80729,0
C00877=36336,35704,-115459,81992,-123751,-80588,0
C00878=35719,36177,-114477,82667,-123430,-80280,0
C00879=36593,36753,-113300,82068,-124258,-80130,0
C00880=42325,30641,-125828,74989,-126250,-83806,0
C00881=39956,29086,-128896,76849,-124151,-84081,0
C00882=35609,33706,-119539,82098,-122629,-81413,0
C00883=35426,33597,-119758,82233,-122466,-81439,0
C00884=35088,34016,-118899,82643,-122341,-81201,0
C00885=35271,34125,-118679,82509,-122505,-81176,0
C00886=34346,35325,-116211,83637,-122160,-80498,0
C00887=35249,35878,-115086,82996,-122991,-80357,0
C00888=35012,36192,-114436,83288,-122902,-80178,0
C00889=35481,36490,-113828,82962,-123341,-80099,0
C00890=35665,36248,-114330,82735,-123409,-80239,0
C00891=36227,35832,-115194,82125,-123708,-80513,0
C00892=36192,35122,-116650,81958,-123471,-80839,0
C00893=40281,30669,-125742,76960,-124907,-83456,0
C00894=40281,30616,-125734,76980,-124934,-83423,0
C00895=36414,35707,-115349,81956,-123843,-80545,0
C00896=41094,30652,-125674,76214,-125488,-83539,0
C00897=40086,29994,-126975,76997,-124591,-83659,0
C00898=35450,35093,-116594,82637,-122948,-80698,0
C00899=36336,35656,-115452,82011,-123771,-80558,0
C00900=35719,36130,-114470,82685,-123448,-80250,0
C00901=36594,36706,-113293,82086,-124277,-80099,0
C00902=42325,30588,-125820,75011,-126278,-83773,0
C00903=39956,29031,-128888,76869,-124179,-84047,0
C00904=35609,33656,-119531,82115,-122649,-81382,0
C00905=35426,33547,-119751,82251,-122485,-81407,0
C00906=35089,33967,-118890,82661,-122361,-81170,0
C00907=35271,34076,-118672,82527,-122524,-81144,0
C00908=34346,35277,-116204,83654,-122178,-80467,0
C00909=35249,35830,-115079,83013,-123009,-80327,0
C00910=35013,36145,-114429,83305,-122921,-80148,0
C00911=35482,36443,-113821,82980,-123360,-80069,0
C00912=35665,36201,-114323,82752,-123428,-80209,0
C00913=36227,35784,-115186,82143,-123727,-80482,0
C00914=36192,35074,-116643,81976,-123491,-80809,0
C00915=40281,30616,-125734,76980,-124934,-83423,0
C00916=40281,30563,-125727,77001,-124960,-83390,0
C00917=36415,35659,-115341,81974,-123863,-80515,0
C00918=41094,30599,-125666,76235,-125514,-83506,0
C00919=40087,29940,-126968,77018,-124618,-83626,0
C00920=35451,35045,-116586,82655,-122968,-80668,0
C00921=36337,35608,-115444,82029,-123790,-80528,0
C00922=35720,36083,-114462,82703,-123468,-80220,0
C00923=36594,36660,-113286,82104,-124296,-80070,0
C00924=42326,30535,-125813,75033,-126307,-83741,0
C00925=39956,28976,-128880,76890,-124206,-84013,0
C00926=35610,33607,-119524,82133,-122669,-81350,0
C00927=35427,33497,-119743,82269,-122506,-81375,0
C00928=35089,33918,-118884,82678,-122380,-81139,0
C00929=35271,34027,-118664,82544,-122544,-81113,0
C00930=34346,35229,-116197,83671,-122197,-80437,0
C00931=35249,35783,-115072,83031,-123027,-80296,0
C00932=35013,36098,-114422,83322,-122939,-80117,0
C00933=35482,36396,-113814,82997,-123378,-80040,0
C00934=35665,36154,-114315,82770,-123447,-80179,0
C00935=36228,35737,-115179,82161,-123747,-80452,0
C00936=36192,35026,-116636,81994,-123511,-80778,0
C00937=40281,30563,-125727,77001,-124960,-83390,0
C00938=40282,30511,-125719,77021,-124987,-83357,0
C00939=36415,35612,-115334,81992,-123884,-80484,0
C00940=41094,30547,-125659,76256,-125542,-83474,0
C00941=40087,29887,-126960,77038,-124644,-83593,0
C00942=35451,34997,-116580,82672,-122986,-80637,0
C00943=36337,35561,-115437,82047,-123810,-80497,0
C00944=35720,36036,-114455,82720,-123486,-80189,0
C00945=36594,36613,-113278,82123,-124316,-80040,0
C00946=42326,30483,-125805,75054,-126335,-83708,0
C00947=39957,28922,-128872,76910,-124234,-83980,0
C00948=35610,33557,-119516,82151,-122690,-81319,0
C00949=35427,33448,-119736,82286,-122525,-81344,0
C00950=35090,33869,-118876,82695,-122400,-81107,0
C00951=35272,33978,-118657,82562,-122564,-81082,0
C00952=34347,35181,-116189,83688,-122215,-80406,0
C00953=35250,35736,-115064,83048,-123047,-80266,0
C00954=35013,36051,-114414,83339,-122957,-80087,0
C00955=35482,36350,-113806,83015,-123396,-80009,0
C00956=35666,36107,-114308,82788,-123465,-80149,0
C00957=36228,35690,-115172,82179,-123766,-80421,0
C00958=36193,34978,-116628,82012,-123531,-80748,0
C00959=40282,30511,-125719,77021,-124987,-83357,0
C00960=40282,30458,-125711,77042,-125013,-83325,0
C00961=36415,35565,-115326,82011,-123903,-80454,0
C00962=41095,30494,-125651,76277,-125568,-83441,0
C00963=40088,29833,-126952,77059,-124672,-83560,0
C00964=35451,34949,-116571,82690,-123006,-80606,0
C00965=36337,35514,-115429,82065,-123830,-80466,0
C00966=35720,35989,-114447,82738,-123504,-80159,0
C00967=36595,36567,-113271,82141,-124335,-80009,0
C00968=42326,30430,-125797,75076,-126363,-83675,0
C00969=39957,28867,-128864,76931,-124260,-83946,0
C00970=35610,33508,-119509,82168,-122710,-81288,0
C00971=35427,33398,-119728,82304,-122546,-81313,0
C00972=35090,33820,-118869,82713,-122420,-81076,0
C00973=35272,33929,-118649,82579,-122584,-81050,0
C00974=34347,35133,-116181,83705,-122233,-80375,0
C00975=35250,35689,-115057,83066,-123065,-80235,0
C00976=35014,36004,-114407,83357,-122976,-80056,0
C00977=35483,36303,-113799,83032,-123415,-79979,0
C00978=35666,36060,-114300,82805,-123485,-80118,0
C00979=36228,35642,-115164,82197,-123786,-80391,0
C00980=36193,34930,-116620,82030,-123550,-80717,0
C00981=40282,30458,-125711,77042,-125013,-83325,0
C00982=40283,30405,-125703,77063,-125040,-83291,0
C00983=36416,35517,-115319,82029,-123923,-80423,0
C00984=41095,30441,-125643,76298,-125596,-83408,0
C00985=40088,29780,-126944,77079,-124698,-83526,0
C00986=37253,32723,-121012,80510,-123693,-81817,0
C00987=37578,32928,-120602,80269,-123987,-81772,0
C00988=35770,35101,-116160,82482,-123319,-80527,0
C00989=36338,35466,-115421,82083,-123849,-80436,0
C00990=35721,35942,-114440,82756,-123524,-80129,0
C00991=36595,36520,-113263,82159,-124354,-79980,0
C00992=42327,30377,-125789,75098,-126392,-83643,0
C00993=39958,28813,-128856,76951,-124288,-83912,0
C00994=36094,32874,-120691,81601,-122910,-81585,0
C00995=36423,33074,-120291,81356,-123204,-81541,0
C00996=34956,34899,-116563,83141,-122656,-80510,0
C00997=34634,34703,-116958,83373,-122362,-80558,0
C00998=34347,35086,-116174,83722,-122252,-80344,0
C00999=35250,35641,-115049,83083,-123084,-80205,0
C01000=35014,35957,-114399,83374,-122994,-80026,0
C01001=35483,36256,-113791,83050,-123433,-79949,0
C01002=35666,36013,-114293,82823,-123503,-80088,0
C01003=36229,35595,-115156,82215,-123805,-80361,0
C01004=38028,32725,-121018,79803,-124243,-81930,0
C01005=40283,30405,-125703,77063,-125040,-83291,0
C01006=40283,30353,-125695,77083,-125066,-83259,0
C01007=36416,35470,-115311,82047,-123942,-80392,0
C01008=41096,30389,-125635,76320,-125623,-83375,0
C01009=40088,29727,-126936,77100,-124725,-83493,0
C01010=37254,32673,-121004,80529,-123715,-81785,0
C01011=37579,32878,-120594,80288,-124010,-81740,0
C01012=35770,35053,-116153,82499,-123339,-80496,0
C01013=36338,35419,-115414,82101,-123869,-80405,0
C01014=35721,35895,-114432,82774,-123542,-80098,0
C01015=36595,36474,-113256,82178,-124373,-79950,0
C01016=47210,22412,-141157,88396,-114327,-84910,0
C01017=39958,28758,-128848,76972,-124316,-83878,0
C01018=36094,32824,-120683,81619,-122931,-81554,0
C01019=36423,33024,-120283,81375,-123225,-81510,0
C01020=34957,34851,-116555,83159,-122675,-80480,0
C01021=34634,34655,-116950,83390,-122380,-80527,0
C01022=34348,35038,-116166,83739,-122270,-80314,0
C01023=35251,35594,-115041,83100,-123102,-80174,0
C01024=35014,35910,-114391,83391,-123013,-79996,0
C01025=35483,36210,-113783,83068,-123451,-79919,0
C01026=35667,35966,-114285,82841,-123522,-80058,0
C01027=36229,35548,-115149,82233,-123825,-80330,0
C01028=38028,32675,-121011,79822,-124266,-81898,0
C01029=40283,30353,-125695,77083,-125066,-83259,0
C01030=40284,30300,-125687,77104,-125092,-83226,0
C01031=36417,35423,-115303,82065,-123962,-80362,0
C01032=41096,30336,-125627,76341,-125650,-83343,0
C01033=40089,29673,-126928,77120,-124751,-83460,0
C01034=37254,32623,-120996,80548,-123736,-81753,0
C01035=37579,32828,-120585,80307,-124032,-81709,0
C01036=35770,35006,-116145,82517,-123358,-80465,0
C01037=36338,35372,-115406,82119,-123888,-80375,0
C01038=35721,35848,-114424,82792,-123562,-80068,0
C01039=36596,36428,-113248,82196,-124393,-79920,0
C01040=47211,22349,-141147,88408,-114346,-84869,0
C01041=39958,28704,-128840,76992,-124343,-83844,0
C01042=36095,32774,-120675,81637,-122952,-81522,0
C01043=36423,32974,-120275,81393,-123247,-81478,0
C01044=34957,34803,-116547,83176,-122693,-80449,0
C01045=34635,34607,-116942,83407,-122399,-80496,0
C01046=34348,34990,-116158,83756,-122289,-80283,0
C01047=35251,35547,-115034,83118,-123122,-80144,0
C01048=35015,35863,-114384,83409,-123030,-79965,0
C01049=35484,36163,-113776,83085,-123471,-79889,0
C01050=35667,35919,-114277,82859,-123541,-80027,0
C01051=36229,35501,-115141,82251,-123844,-80300,0
C01052=38029,32625,-121003,79841,-124289,-81866,0
C01053=40284,30300,-125687,77104,-125092,-83226,0
C01054=40284,30248,-125679,77125,-125119,-83193,0
C01055=36417,35376,-115295,82084,-123981,-80332,0
C01056=41096,30284,-125619,76362,-125677,-83309,0
C01057=40089,29620,-126920,77141,-124779,-83427,0
C01058=37254,32573,-120988,80566,-123759,-81721,0
C01059=37579,32778,-120577,80327,-124054,-81677,0
C01060=35771,34958,-116137,82535,-123377,-80434,0
C01061=36339,35324,-115398,82138,-123908,-80344,0
C01062=35722,35801,-114416,82809,-123580,-80038,0
C01063=36596,36381,-113240,82214,-124411,-79889,0
C01064=47211,22285,-141138,88421,-114364,-84829,0
C01065=39959,28649,-128832,77013,-124371,-83811,0
C01066=36095,32724,-120667,81655,-122972,-81490,0
C01067=36424,32925,-120267,81411,-123268,-81446,0
C01068=34957,34755,-116539,83193,-122713,-80417,0
C01069=34635,34559,-116933,83424,-122417,-80465,0
C01070=34348,34943,-116150,83773,-122307,-80252,0
C01071=35251,35500,-115026,83136,-123140,-80113,0
C01072=35015,35816,-114376,83426,-123048,-79935,0
C01073=35484,36117,-113768,83103,-123489,-79858,0
C01074=35667,35873,-114269,82876,-123560,-79997,0
C01075=36230,35454,-115133,82270,-123864,-80269,0
C01076=38029,32575,-120995,79861,-124311,-81834,0
C01077=40284,30248,-125679,77125,-125119,-83193,0
C01078=40284,30195,-125671,77145,-125145,-83160,0
C01079=36417,35328,-115287,82102,-124001,-80301,0
C01080=41097,30231,-125611,76383,-125704,-83277,0
C01081=40090,29567,-126910,77162,-124805,-83394,0
C01082=37255,32523,-120980,80585,-123781,-81689,0
C01083=37580,32729,-120569,80346,-124075,-81645,0
C01084=35771,34911,-116129,82553,-123396,-80403,0
C01085=36339,35277,-115390,82156,-123927,-80314,0
C01086=35722,35754,-114409,82827,-123600,-80007,0
C01087=36596,36335,-113232,82233,-124431,-79859,0
C01088=47212,22222,-141129,88433,-114383,-84789,0
C01089=39959,28595,-128824,77034,-124398,-83777,0
C01090=36095,32674,-120659,81673,-122994,-81458,0
C01091=36424,32875,-120259,81430,-123289,-81414,0
C01092=34958,34708,-116531,83211,-122731,-80387,0
C01093=34635,34511,-116925,83441,-122437,-80434,0
C01094=34349,34895,-116142,83790,-122325,-80221,0
C01095=35252,35453,-115018,83153,-123158,-80083,0
C01096=35015,35770,-114368,83443,-123067,-79904,0
C01097=35484,36070,-113760,83121,-123508,-79828,0
C01098=35668,35826,-114261,82894,-123578,-79967,0
C01099=36230,35407,-115125,82288,-123884,-80239,0
C01100=38030,32525,-120987,79880,-124334,-81802,0
C01101=40284,30195,-125671,77145,-125145,-83160,0
C01102=40285,30143,-125662,77166,-125172,-83127,0
C01103=36418,35281,-115279,82120,-124020,-80271,0
C01104=41097,30179,-125602,76404,-125731,-83244,0
C01105=40090,29514,-126902,77183,-124832,-83360,0
C01106=37255,32473,-120972,80604,-123803,-81657,0
C01107=37580,32679,-120561,80365,-124098,-81613,0
C01108=35771,34863,-116121,82571,-123416,-80372,0
C01109=36340,35230,-115382,82174,-123947,-80283,0
C01110=35722,35707,-114401,82845,-123618,-79977,0
C01111=36597,36289,-113224,82251,-124450,-79829,0
C01112=47212,22158,-141119,88446,-114401,-84749,0
C01113=39960,28541,-128815,77054,-124425,-83743,0
C01114=36096,32625,-120651,81691,-123015,-81427,0
C01115=36424,32826,-120251,81448,-123310,-81383,0
C01116=34958,34660,-116523,83228,-122750,-80356,0
C01117=34636,34464,-116917,83459,-122455,-80403,0
C01118=34349,34848,-116134,83807,-122344,-80191,0
C01119=35252,35406,-115010,83171,-123177,-80052,0
C01120=35016,35723,-114360,83461,-123085,-79874,0
C01121=35485,36024,-113752,83139,-123526,-79798,0
C01122=35668,35779,-114253,82912,-123597,-79936,0
C01123=36230,35360,-115117,82306,-123903,-80208,0
C01124=38030,32475,-120977,79900,-124357,-81770,0
C01125=40285,30143,-125662,77166,-125172,-83127,0
C01126=40285,30090,-125653,77187,-125198,-83094,0
C01127=36418,35234,-115271,82139,-124040,-80240,0
C01128=41098,30127,-125594,76426,-125758,-83211,0
C01129=40091,29461,-126894,77203,-124858,-83327,0
C01130=37255,32423,-120964,80623,-123825,-81626,0
C01131=37580,32630,-120553,80384,-124120,-81581,0
C01132=35772,34816,-116113,82589,-123435,-80341,0
C01133=36340,35183,-115374,82193,-123966,-80253,0
C01134=35723,35661,-114392,82863,-123636,-79946,0
C01135=36597,36243,-113216,82270,-124470,-79799,0
C01136=47213,22095,-141109,88459,-114420,-84708,0
C01137=39960,28486,-128807,77075,-124452,-83709,0
//INST
///DATE 2025/02/20 16:20
///COMM Generated using RoboDK
///ATTR SC,RW
///GROUP1 RB1
NOP
MOVL C00000 V=130.0 PL=1
CALL JOB:EXTRUDE
MOVL C00001 V=30.0 PL=1
CALL JOB:EXTRUDE
MOVL C00002 V=30.0 PL=1
CALL JOB:EXTRUDE
MOVL C00003 V=30.0 PL=1
CALL JOB:EXTRUDE
MOVL C00004 V=30.0 PL=1
CALL JOB:EXTRUDE
MOVL C00005 V=30.0 PL=1
CALL JOB:EXTRUDE
MOVL C00006 V=30.0 PL=1
CALL JOB:EXTRUDE
MOVL C00007 V=30.0 PL=1
CALL JOB:EXTRUDE
MOVL C00008 V=30.0 PL=1
MOVL C00009 V=130.0 PL=1
MOVL C00010 V=130.0 PL=1
CALL JOB:EXTRUDE
MOVL C00011 V=20.0 PL=1
MOVL C00012 V=130.0 PL=1
MOVL C00013 V=130.0 PL=1
CALL JOB:EXTRUDE
MOVL C00014 V=60.0 PL=1
CALL JOB:EXTRUDE
MOVL C00015 V=60.0 PL=1
CALL JOB:EXTRUDE
MOVL C00016 V=60.0 PL=1
CALL JOB:EXTRUDE
MOVL C00017 V=60.0 PL=1
MOVL C00018 V=130.0 PL=1
CALL JOB:EXTRUDE
MOVL C00019 V=30.0 PL=1
CALL JOB:EXTRUDE
MOVL C00020 V=30.0 PL=1
CALL JOB:EXTRUDE
MOVL C00021 V=30.0 PL=1
CALL JOB:EXTRUDE
MOVL C00022 V=30.0 PL=1
CALL JOB:EXTRUDE
MOVL C00023 V=30.0 PL=1
CALL JOB:EXTRUDE
MOVL C00024 V=30.0 PL=1
CALL JOB:EXTRUDE
MOVL C00025 V=30.0 PL=1
CALL JOB:EXTRUDE
MOVL C00026 V=30.0 PL=1
MOVL C00027 V=130.0 PL=1
MOVL C00028 V=130.0 PL=1
CALL JOB:EXTRUDE
MOVL C00029 V=20.0 PL=1
MOVL C00030 V=130.0 PL=1
MOVL C00031 V=130.0 PL=1
CALL JOB:EXTRUDE
MOVL C00032 V=60.0 PL=1
CALL JOB:EXTRUDE
MOVL C00033 V=60.0 PL=1
CALL JOB:EXTRUDE
MOVL C00034 V=60.0 PL=1
CALL JOB:EXTRUDE
MOVL C00035 V=60.0 PL=1
MOVL C00036 V=130.0 PL=1
CALL JOB:EXTRUDE
MOVL C00037 V=30.0 PL=1
CALL JOB:EXTRUDE
MOVL C00038 V=30.0 PL=1
CALL JOB:EXTRUDE
MOVL C00039 V=30.0 PL=1
CALL JOB:EXTRUDE
MOVL C00040 V=30.0 PL=1
CALL JOB:EXTRUDE
MOVL C00041 V=30.0 PL=1
CALL JOB:EXTRUDE
MOVL C00042 V=30.0 PL=1
CALL JOB:EXTRUDE
MOVL C00043 V=30.0 PL=1
CALL JOB:EXTRUDE
MOVL C00044 V=30.0 PL=1
MOVL C00045 V=130.0 PL=1
MOVL C00046 V=130.0 PL=1
CALL JOB:EXTRUDE
MOVL C00047 V=20.0 PL=1
MOVL C00048 V=130.0 PL=1
MOVL C00049 V=130.0 PL=1
CALL JOB:EXTRUDE
MOVL C00050 V=60.0 PL=1
CALL JOB:EXTRUDE
MOVL C00051 V=60.0 PL=1
CALL JOB:EXTRUDE
MOVL C00052 V=60.0 PL=1
CALL JOB:EXTRUDE
MOVL C00053 V=60.0 PL=1
MOVL C00054 V=130.0 PL=1
CALL JOB:EXTRUDE
MOVL C00055 V=30.0 PL=1
CALL JOB:EXTRUDE
MOVL C00056 V=30.0 PL=1
CALL JOB:EXTRUDE
MOVL C00057 V=30.0 PL=1
CALL JOB:EXTRUDE
MOVL C00058 V=30.0 PL=1
CALL JOB:EXTRUDE
MOVL C00059 V=30.0 PL=1
CALL JOB:EXTRUDE
MOVL C00060 V=30.0 PL=1
CALL JOB:EXTRUDE
MOVL C00061 V=30.0 PL=1
CALL JOB:EXTRUDE
MOVL C00062 V=30.0 PL=1
MOVL C00063 V=130.0 PL=1
MOVL C00064 V=130.0 PL=1
CALL JOB:EXTRUDE
MOVL C00065 V=20.0 PL=1
MOVL C00066 V=130.0 PL=1
MOVL C00067 V=130.0 PL=1
CALL JOB:EXTRUDE
MOVL C00068 V=60.0 PL=1
CALL JOB:EXTRUDE
MOVL C00069 V=60.0 PL=1
CALL JOB:EXTRUDE
MOVL C00070 V=60.0 PL=1
CALL JOB:EXTRUDE
MOVL C00071 V=60.0 PL=1
MOVL C00072 V=130.0 PL=1
CALL JOB:EXTRUDE
MOVL C00073 V=30.0 PL=1
CALL JOB:EXTRUDE
MOVL C00074 V=30.0 PL=1
CALL JOB:EXTRUDE
MOVL C00075 V=30.0 PL=1
CALL JOB:EXTRUDE
MOVL C00076 V=30.0 PL=1
CALL JOB:EXTRUDE
MOVL C00077 V=30.0 PL=1
CALL JOB:EXTRUDE
MOVL C00078 V=30.0 PL=1
CALL JOB:EXTRUDE
MOVL C00079 V=30.0 PL=1
CALL JOB:EXTRUDE
MOVL C00080 V=30.0 PL=1
MOVL C00081 V=130.0 PL=1
MOVL C00082 V=130.0 PL=1
CALL JOB:EXTRUDE
MOVL C00083 V=20.0 PL=1
MOVL C00084 V=130.0 PL=1
MOVL C00085 V=130.0 PL=1
CALL JOB:EXTRUDE
MOVL C00086 V=60.0 PL=1
CALL JOB:EXTRUDE
MOVL C00087 V=60.0 PL=1
CALL JOB:EXTRUDE
MOVL C00088 V=60.0 PL=1
CALL JOB:EXTRUDE
MOVL C00089 V=60.0 PL=1
MOVL C00090 V=130.0 PL=1
CALL JOB:EXTRUDE
MOVL C00091 V=30.0 PL=1
CALL JOB:EXTRUDE
MOVL C00092 V=30.0 PL=1
CALL JOB:EXTRUDE
MOVL C00093 V=30.0 PL=1
CALL JOB:EXTRUDE
MOVL C00094 V=30.0 PL=1
CALL JOB:EXTRUDE
MOVL C00095 V=30.0 PL=1
CALL JOB:EXTRUDE
MOVL C00096 V=30.0 PL=1
CALL JOB:EXTRUDE
MOVL C00097 V=30.0 PL=1
CALL JOB:EXTRUDE
MOVL C00098 V=30.0 PL=1
MOVL C00099 V=130.0 PL=1
MOVL C00100 V=130.0 PL=1
CALL JOB:EXTRUDE
MOVL C00101 V=20.0 PL=1
MOVL C00102 V=130.0 PL=1
MOVL C00103 V=130.0 PL=1
CALL JOB:EXTRUDE
MOVL C00104 V=60.0 PL=1
CALL JOB:EXTRUDE
MOVL C00105 V=60.0 PL=1
CALL JOB:EXTRUDE
MOVL C00106 V=60.0 PL=1
CALL JOB:EXTRUDE
MOVL C00107 V=60.0 PL=1
MOVL C00108 V=130.0 PL=1
CALL JOB:EXTRUDE
MOVL C00109 V=30.0 PL=1
CALL JOB:EXTRUDE
MOVL C00110 V=30.0 PL=1
CALL JOB:EXTRUDE
MOVL C00111 V=30.0 PL=1
CALL JOB:EXTRUDE
MOVL C00112 V=30.0 PL=1
CALL JOB:EXTRUDE
MOVL C00113 V=30.0 PL=1
CALL JOB:EXTRUDE
MOVL C00114 V=30.0 PL=1
CALL JOB:EXTRUDE
MOVL C00115 V=30.0 PL=1
CALL JOB:EXTRUDE
MOVL C00116 V=30.0 PL=1
MOVL C00117 V=130.0 PL=1
MOVL C00118 V=130.0 PL=1
CALL JOB:EXTRUDE
MOVL C00119 V=20.0 PL=1
MOVL C00120 V=130.0 PL=1
MOVL C00121 V=130.0 PL=1
CALL JOB:EXTRUDE
MOVL C00122 V=60.0 PL=1
CALL JOB:EXTRUDE
MOVL C00123 V=60.0 PL=1
CALL JOB:EXTRUDE
MOVL C00124 V=60.0 PL=1
CALL JOB:EXTRUDE
MOVL C00125 V=60.0 PL=1
MOVL C00126 V=130.0 PL=1
CALL JOB:EXTRUDE
MOVL C00127 V=30.0 PL=1
CALL JOB:EXTRUDE
MOVL C00128 V=30.0 PL=1
CALL JOB:EXTRUDE
MOVL C00129 V=30.0 PL=1
CALL JOB:EXTRUDE
MOVL C00130 V=30.0 PL=1
CALL JOB:EXTRUDE
MOVL C00131 V=30.0 PL=1
CALL JOB:EXTRUDE
MOVL C00132 V=30.0 PL=1
CALL JOB:EXTRUDE
MOVL C00133 V=30.0 PL=1
CALL JOB:EXTRUDE
MOVL C00134 V=30.0 PL=1
MOVL C00135 V=130.0 PL=1
MOVL C00136 V=130.0 PL=1
CALL JOB:EXTRUDE
MOVL C00137 V=20.0 PL=1
MOVL C00138 V=130.0 PL=1
MOVL C00139 V=130.0 PL=1
CALL JOB:EXTRUDE
MOVL C00140 V=60.0 PL=1
CALL JOB:EXTRUDE
MOVL C00141 V=60.0 PL=1
CALL JOB:EXTRUDE
MOVL C00142 V=60.0 PL=1
CALL JOB:EXTRUDE
MOVL C00143 V=60.0 PL=1
MOVL C00144 V=130.0 PL=1
CALL JOB:EXTRUDE
MOVL C00145 V=30.0 PL=1
CALL JOB:EXTRUDE
MOVL C00146 V=30.0 PL=1
CALL JOB:EXTRUDE
MOVL C00147 V=30.0 PL=1
CALL JOB:EXTRUDE
MOVL C00148 V=30.0 PL=1
CALL JOB:EXTRUDE
MOVL C00149 V=30.0 PL=1
CALL JOB:EXTRUDE
MOVL C00150 V=30.0 PL=1
CALL JOB:EXTRUDE
MOVL C00151 V=30.0 PL=1
CALL JOB:EXTRUDE
MOVL C00152 V=30.0 PL=1
MOVL C00153 V=130.0 PL=1
MOVL C00154 V=130.0 PL=1
CALL JOB:EXTRUDE
MOVL C00155 V=20.0 PL=1
MOVL C00156 V=130.0 PL=1
MOVL C00157 V=130.0 PL=1
CALL JOB:EXTRUDE
MOVL C00158 V=60.0 PL=1
CALL JOB:EXTRUDE
MOVL C00159 V=60.0 PL=1
CALL JOB:EXTRUDE
MOVL C00160 V=60.0 PL=1
CALL JOB:EXTRUDE
MOVL C00161 V=60.0 PL=1
MOVL C00162 V=130.0 PL=1
CALL JOB:EXTRUDE
MOVL C00163 V=30.0 PL=1
CALL JOB:EXTRUDE
MOVL C00164 V=30.0 PL=1
CALL JOB:EXTRUDE
MOVL C00165 V=30.0 PL=1
CALL JOB:EXTRUDE
MOVL C00166 V=30.0 PL=1
CALL JOB:EXTRUDE
MOVL C00167 V=30.0 PL=1
CALL JOB:EXTRUDE
MOVL C00168 V=30.0 PL=1
CALL JOB:EXTRUDE
MOVL C00169 V=30.0 PL=1
CALL JOB:EXTRUDE
MOVL C00170 V=30.0 PL=1
MOVL C00171 V=130.0 PL=1
MOVL C00172 V=130.0 PL=1
CALL JOB:EXTRUDE
MOVL C00173 V=20.0 PL=1
MOVL C00174 V=130.0 PL=1
MOVL C00175 V=130.0 PL=1
CALL JOB:EXTRUDE
MOVL C00176 V=60.0 PL=1
CALL JOB:EXTRUDE
MOVL C00177 V=60.0 PL=1
CALL JOB:EXTRUDE
MOVL C00178 V=60.0 PL=1
CALL JOB:EXTRUDE
MOVL C00179 V=60.0 PL=1
MOVL C00180 V=130.0 PL=1
CALL JOB:EXTRUDE
MOVL C00181 V=30.0 PL=1
CALL JOB:EXTRUDE
MOVL C00182 V=30.0 PL=1
CALL JOB:EXTRUDE
MOVL C00183 V=30.0 PL=1
CALL JOB:EXTRUDE
MOVL C00184 V=30.0 PL=1
CALL JOB:EXTRUDE
MOVL C00185 V=30.0 PL=1
CALL JOB:EXTRUDE
MOVL C00186 V=30.0 PL=1
CALL JOB:EXTRUDE
MOVL C00187 V=30.0 PL=1
CALL JOB:EXTRUDE
MOVL C00188 V=30.0 PL=1
MOVL C00189 V=130.0 PL=1
MOVL C00190 V=130.0 PL=1
CALL JOB:EXTRUDE
MOVL C00191 V=20.0 PL=1
MOVL C00192 V=130.0 PL=1
MOVL C00193 V=130.0 PL=1
CALL JOB:EXTRUDE
MOVL C00194 V=60.0 PL=1
CALL JOB:EXTRUDE
MOVL C00195 V=60.0 PL=1
CALL JOB:EXTRUDE
MOVL C00196 V=60.0 PL=1
CALL JOB:EXTRUDE
MOVL C00197 V=60.0 PL=1
MOVL C00198 V=130.0 PL=1
CALL JOB:EXTRUDE
MOVL C00199 V=30.0 PL=1
CALL JOB:EXTRUDE
MOVL C00200 V=30.0 PL=1
CALL JOB:EXTRUDE
MOVL C00201 V=30.0 PL=1
CALL JOB:EXTRUDE
MOVL C00202 V=30.0 PL=1
CALL JOB:EXTRUDE
MOVL C00203 V=30.0 PL=1
CALL JOB:EXTRUDE
MOVL C00204 V=30.0 PL=1
CALL JOB:EXTRUDE
MOVL C00205 V=30.0 PL=1
CALL JOB:EXTRUDE
MOVL C00206 V=30.0 PL=1
MOVL C00207 V=130.0 PL=1
MOVL C00208 V=130.0 PL=1
CALL JOB:EXTRUDE
MOVL C00209 V=20.0 PL=1
MOVL C00210 V=130.0 PL=1
MOVL C00211 V=130.0 PL=1
CALL JOB:EXTRUDE
MOVL C00212 V=60.0 PL=1
CALL JOB:EXTRUDE
MOVL C00213 V=60.0 PL=1
CALL JOB:EXTRUDE
MOVL C00214 V=60.0 PL=1
CALL JOB:EXTRUDE
MOVL C00215 V=60.0 PL=1
MOVL C00216 V=130.0 PL=1
CALL JOB:EXTRUDE
MOVL C00217 V=30.0 PL=1
CALL JOB:EXTRUDE
MOVL C00218 V=30.0 PL=1
CALL JOB:EXTRUDE
MOVL C00219 V=30.0 PL=1
CALL JOB:EXTRUDE
MOVL C00220 V=30.0 PL=1
CALL JOB:EXTRUDE
MOVL C00221 V=30.0 PL=1
CALL JOB:EXTRUDE
MOVL C00222 V=30.0 PL=1
CALL JOB:EXTRUDE
MOVL C00223 V=30.0 PL=1
CALL JOB:EXTRUDE
MOVL C00224 V=30.0 PL=1
MOVL C00225 V=130.0 PL=1
MOVL C00226 V=130.0 PL=1
CALL JOB:EXTRUDE
MOVL C00227 V=20.0 PL=1
MOVL C00228 V=130.0 PL=1
MOVL C00229 V=130.0 PL=1
CALL JOB:EXTRUDE
MOVL C00230 V=60.0 PL=1
CALL JOB:EXTRUDE
MOVL C00231 V=60.0 PL=1
CALL JOB:EXTRUDE
MOVL C00232 V=60.0 PL=1
CALL JOB:EXTRUDE
MOVL C00233 V=60.0 PL=1
MOVL C00234 V=130.0 PL=1
CALL JOB:EXTRUDE
MOVL C00235 V=30.0 PL=1
CALL JOB:EXTRUDE
MOVL C00236 V=30.0 PL=1
CALL JOB:EXTRUDE
MOVL C00237 V=30.0 PL=1
CALL JOB:EXTRUDE
MOVL C00238 V=30.0 PL=1
CALL JOB:EXTRUDE
MOVL C00239 V=30.0 PL=1
CALL JOB:EXTRUDE
MOVL C00240 V=30.0 PL=1
CALL JOB:EXTRUDE
MOVL C00241 V=30.0 PL=1
CALL JOB:EXTRUDE
MOVL C00242 V=30.0 PL=1
MOVL C00243 V=130.0 PL=1
MOVL C00244 V=130.0 PL=1
CALL JOB:EXTRUDE
MOVL C00245 V=20.0 PL=1
MOVL C00246 V=130.0 PL=1
MOVL C00247 V=130.0 PL=1
CALL JOB:EXTRUDE
MOVL C00248 V=60.0 PL=1
CALL JOB:EXTRUDE
MOVL C00249 V=60.0 PL=1
CALL JOB:EXTRUDE
MOVL C00250 V=60.0 PL=1
CALL JOB:EXTRUDE
MOVL C00251 V=60.0 PL=1
MOVL C00252 V=130.0 PL=1
CALL JOB:EXTRUDE
MOVL C00253 V=30.0 PL=1
CALL JOB:EXTRUDE
MOVL C00254 V=30.0 PL=1
CALL JOB:EXTRUDE
MOVL C00255 V=30.0 PL=1
CALL JOB:EXTRUDE
MOVL C00256 V=30.0 PL=1
CALL JOB:EXTRUDE
MOVL C00257 V=30.0 PL=1
CALL JOB:EXTRUDE
MOVL C00258 V=30.0 PL=1
CALL JOB:EXTRUDE
MOVL C00259 V=30.0 PL=1
CALL JOB:EXTRUDE
MOVL C00260 V=30.0 PL=1
MOVL C00261 V=130.0 PL=1
MOVL C00262 V=130.0 PL=1
CALL JOB:EXTRUDE
MOVL C00263 V=20.0 PL=1
MOVL C00264 V=130.0 PL=1
MOVL C00265 V=130.0 PL=1
CALL JOB:EXTRUDE
MOVL C00266 V=60.0 PL=1
CALL JOB:EXTRUDE
MOVL C00267 V=60.0 PL=1
CALL JOB:EXTRUDE
MOVL C00268 V=60.0 PL=1
CALL JOB:EXTRUDE
MOVL C00269 V=60.0 PL=1
MOVL C00270 V=130.0 PL=1
CALL JOB:EXTRUDE
MOVL C00271 V=30.0 PL=1
CALL JOB:EXTRUDE
MOVL C00272 V=30.0 PL=1
CALL JOB:EXTRUDE
MOVL C00273 V=30.0 PL=1
CALL JOB:EXTRUDE
MOVL C00274 V=30.0 PL=1
CALL JOB:EXTRUDE
MOVL C00275 V=30.0 PL=1
CALL JOB:EXTRUDE
MOVL C00276 V=30.0 PL=1
CALL JOB:EXTRUDE
MOVL C00277 V=30.0 PL=1
CALL JOB:EXTRUDE
MOVL C00278 V=30.0 PL=1
MOVL C00279 V=130.0 PL=1
MOVL C00280 V=130.0 PL=1
CALL JOB:EXTRUDE
MOVL C00281 V=20.0 PL=1
MOVL C00282 V=130.0 PL=1
MOVL C00283 V=130.0 PL=1
CALL JOB:EXTRUDE
MOVL C00284 V=60.0 PL=1
CALL JOB:EXTRUDE
MOVL C00285 V=60.0 PL=1
CALL JOB:EXTRUDE
MOVL C00286 V=60.0 PL=1
CALL JOB:EXTRUDE
MOVL C00287 V=60.0 PL=1
MOVL C00288 V=130.0 PL=1
CALL JOB:EXTRUDE
MOVL C00289 V=30.0 PL=1
CALL JOB:EXTRUDE
MOVL C00290 V=30.0 PL=1
CALL JOB:EXTRUDE
MOVL C00291 V=30.0 PL=1
CALL JOB:EXTRUDE
MOVL C00292 V=30.0 PL=1
CALL JOB:EXTRUDE
MOVL C00293 V=30.0 PL=1
CALL JOB:EXTRUDE
MOVL C00294 V=30.0 PL=1
CALL JOB:EXTRUDE
MOVL C00295 V=30.0 PL=1
CALL JOB:EXTRUDE
MOVL C00296 V=30.0 PL=1
MOVL C00297 V=130.0 PL=1
MOVL C00298 V=130.0 PL=1
CALL JOB:EXTRUDE
MOVL C00299 V=20.0 PL=1
MOVL C00300 V=130.0 PL=1
MOVL C00301 V=130.0 PL=1
CALL JOB:EXTRUDE
MOVL C00302 V=60.0 PL=1
CALL JOB:EXTRUDE
MOVL C00303 V=60.0 PL=1
CALL JOB:EXTRUDE
MOVL C00304 V=60.0 PL=1
CALL JOB:EXTRUDE
MOVL C00305 V=60.0 PL=1
MOVL C00306 V=130.0 PL=1
CALL JOB:EXTRUDE
MOVL C00307 V=30.0 PL=1
CALL JOB:EXTRUDE
MOVL C00308 V=30.0 PL=1
CALL JOB:EXTRUDE
MOVL C00309 V=30.0 PL=1
CALL JOB:EXTRUDE
MOVL C00310 V=30.0 PL=1
CALL JOB:EXTRUDE
MOVL C00311 V=30.0 PL=1
CALL JOB:EXTRUDE
MOVL C00312 V=30.0 PL=1
CALL JOB:EXTRUDE
MOVL C00313 V=30.0 PL=1
CALL JOB:EXTRUDE
MOVL C00314 V=30.0 PL=1
MOVL C00315 V=130.0 PL=1
MOVL C00316 V=130.0 PL=1
CALL JOB:EXTRUDE
MOVL C00317 V=20.0 PL=1
MOVL C00318 V=130.0 PL=1
MOVL C00319 V=130.0 PL=1
CALL JOB:EXTRUDE
MOVL C00320 V=60.0 PL=1
CALL JOB:EXTRUDE
MOVL C00321 V=60.0 PL=1
CALL JOB:EXTRUDE
MOVL C00322 V=60.0 PL=1
CALL JOB:EXTRUDE
MOVL C00323 V=60.0 PL=1
MOVL C00324 V=130.0 PL=1
CALL JOB:EXTRUDE
MOVL C00325 V=30.0 PL=1
CALL JOB:EXTRUDE
MOVL C00326 V=30.0 PL=1
CALL JOB:EXTRUDE
MOVL C00327 V=30.0 PL=1
CALL JOB:EXTRUDE
MOVL C00328 V=30.0 PL=1
CALL JOB:EXTRUDE
MOVL C00329 V=30.0 PL=1
CALL JOB:EXTRUDE
MOVL C00330 V=30.0 PL=1
CALL JOB:EXTRUDE
MOVL C00331 V=30.0 PL=1
CALL JOB:EXTRUDE
MOVL C00332 V=30.0 PL=1
MOVL C00333 V=130.0 PL=1
MOVL C00334 V=130.0 PL=1
CALL JOB:EXTRUDE
MOVL C00335 V=20.0 PL=1
MOVL C00336 V=130.0 PL=1
MOVL C00337 V=130.0 PL=1
CALL JOB:EXTRUDE
MOVL C00338 V=60.0 PL=1
CALL JOB:EXTRUDE
MOVL C00339 V=60.0 PL=1
CALL JOB:EXTRUDE
MOVL C00340 V=60.0 PL=1
CALL JOB:EXTRUDE
MOVL C00341 V=60.0 PL=1
MOVL C00342 V=130.0 PL=1
CALL JOB:EXTRUDE
MOVL C00343 V=30.0 PL=1
CALL JOB:EXTRUDE
MOVL C00344 V=30.0 PL=1
CALL JOB:EXTRUDE
MOVL C00345 V=30.0 PL=1
CALL JOB:EXTRUDE
MOVL C00346 V=30.0 PL=1
CALL JOB:EXTRUDE
MOVL C00347 V=30.0 PL=1
CALL JOB:EXTRUDE
MOVL C00348 V=30.0 PL=1
CALL JOB:EXTRUDE
MOVL C00349 V=30.0 PL=1
CALL JOB:EXTRUDE
MOVL C00350 V=30.0 PL=1
MOVL C00351 V=130.0 PL=1
MOVL C00352 V=130.0 PL=1
CALL JOB:EXTRUDE
MOVL C00353 V=20.0 PL=1
MOVL C00354 V=130.0 PL=1
MOVL C00355 V=130.0 PL=1
CALL JOB:EXTRUDE
MOVL C00356 V=60.0 PL=1
CALL JOB:EXTRUDE
MOVL C00357 V=60.0 PL=1
CALL JOB:EXTRUDE
MOVL C00358 V=60.0 PL=1
CALL JOB:EXTRUDE
MOVL C00359 V=60.0 PL=1
MOVL C00360 V=130.0 PL=1
CALL JOB:EXTRUDE
MOVL C00361 V=30.0 PL=1
CALL JOB:EXTRUDE
MOVL C00362 V=30.0 PL=1
CALL JOB:EXTRUDE
MOVL C00363 V=30.0 PL=1
CALL JOB:EXTRUDE
MOVL C00364 V=30.0 PL=1
CALL JOB:EXTRUDE
MOVL C00365 V=30.0 PL=1
CALL JOB:EXTRUDE
MOVL C00366 V=30.0 PL=1
CALL JOB:EXTRUDE
MOVL C00367 V=30.0 PL=1
CALL JOB:EXTRUDE
MOVL C00368 V=30.0 PL=1
MOVL C00369 V=130.0 PL=1
MOVL C00370 V=130.0 PL=1
CALL JOB:EXTRUDE
MOVL C00371 V=20.0 PL=1
MOVL C00372 V=130.0 PL=1
MOVL C00373 V=130.0 PL=1
CALL JOB:EXTRUDE
MOVL C00374 V=60.0 PL=1
CALL JOB:EXTRUDE
MOVL C00375 V=60.0 PL=1
CALL JOB:EXTRUDE
MOVL C00376 V=60.0 PL=1
CALL JOB:EXTRUDE
MOVL C00377 V=60.0 PL=1
MOVL C00378 V=130.0 PL=1
CALL JOB:EXTRUDE
MOVL C00379 V=30.0 PL=1
CALL JOB:EXTRUDE
MOVL C00380 V=30.0 PL=1
CALL JOB:EXTRUDE
MOVL C00381 V=30.0 PL=1
CALL JOB:EXTRUDE
MOVL C00382 V=30.0 PL=1
CALL JOB:EXTRUDE
MOVL C00383 V=30.0 PL=1
CALL JOB:EXTRUDE
MOVL C00384 V=30.0 PL=1
CALL JOB:EXTRUDE
MOVL C00385 V=30.0 PL=1
CALL JOB:EXTRUDE
MOVL C00386 V=30.0 PL=1
MOVL C00387 V=130.0 PL=1
MOVL C00388 V=130.0 PL=1
CALL JOB:EXTRUDE
MOVL C00389 V=20.0 PL=1
MOVL C00390 V=130.0 PL=1
MOVL C00391 V=130.0 PL=1
CALL JOB:EXTRUDE
MOVL C00392 V=60.0 PL=1
CALL JOB:EXTRUDE
MOVL C00393 V=60.0 PL=1
CALL JOB:EXTRUDE
MOVL C00394 V=60.0 PL=1
CALL JOB:EXTRUDE
MOVL C00395 V=60.0 PL=1
MOVL C00396 V=130.0 PL=1
CALL JOB:EXTRUDE
MOVL C00397 V=30.0 PL=1
CALL JOB:EXTRUDE
MOVL C00398 V=30.0 PL=1
CALL JOB:EXTRUDE
MOVL C00399 V=30.0 PL=1
CALL JOB:EXTRUDE
MOVL C00400 V=30.0 PL=1
CALL JOB:EXTRUDE
MOVL C00401 V=30.0 PL=1
CALL JOB:EXTRUDE
MOVL C00402 V=30.0 PL=1
CALL JOB:EXTRUDE
MOVL C00403 V=30.0 PL=1
CALL JOB:EXTRUDE
MOVL C00404 V=30.0 PL=1
MOVL C00405 V=130.0 PL=1
MOVL C00406 V=130.0 PL=1
CALL JOB:EXTRUDE
MOVL C00407 V=20.0 PL=1
MOVL C00408 V=130.0 PL=1
MOVL C00409 V=130.0 PL=1
CALL JOB:EXTRUDE
MOVL C00410 V=60.0 PL=1
CALL JOB:EXTRUDE
MOVL C00411 V=60.0 PL=1
CALL JOB:EXTRUDE
MOVL C00412 V=60.0 PL=1
CALL JOB:EXTRUDE
MOVL C00413 V=60.0 PL=1
MOVL C00414 V=130.0 PL=1
CALL JOB:EXTRUDE
MOVL C00415 V=30.0 PL=1
CALL JOB:EXTRUDE
MOVL C00416 V=30.0 PL=1
CALL JOB:EXTRUDE
MOVL C00417 V=30.0 PL=1
CALL JOB:EXTRUDE
MOVL C00418 V=30.0 PL=1
CALL JOB:EXTRUDE
MOVL C00419 V=30.0 PL=1
CALL JOB:EXTRUDE
MOVL C00420 V=30.0 PL=1
CALL JOB:EXTRUDE
MOVL C00421 V=30.0 PL=1
CALL JOB:EXTRUDE
MOVL C00422 V=30.0 PL=1
MOVL C00423 V=130.0 PL=1
MOVL C00424 V=130.0 PL=1
CALL JOB:EXTRUDE
MOVL C00425 V=20.0 PL=1
MOVL C00426 V=130.0 PL=1
MOVL C00427 V=130.0 PL=1
CALL JOB:EXTRUDE
MOVL C00428 V=60.0 PL=1
CALL JOB:EXTRUDE
MOVL C00429 V=60.0 PL=1
CALL JOB:EXTRUDE
MOVL C00430 V=60.0 PL=1
CALL JOB:EXTRUDE
MOVL C00431 V=60.0 PL=1
MOVL C00432 V=130.0 PL=1
CALL JOB:EXTRUDE
MOVL C00433 V=30.0 PL=1
CALL JOB:EXTRUDE
MOVL C00434 V=30.0 PL=1
CALL JOB:EXTRUDE
MOVL C00435 V=30.0 PL=1
CALL JOB:EXTRUDE
MOVL C00436 V=30.0 PL=1
CALL JOB:EXTRUDE
MOVL C00437 V=30.0 PL=1
CALL JOB:EXTRUDE
MOVL C00438 V=30.0 PL=1
CALL JOB:EXTRUDE
MOVL C00439 V=30.0 PL=1
CALL JOB:EXTRUDE
MOVL C00440 V=30.0 PL=1
MOVL C00441 V=130.0 PL=1
MOVL C00442 V=130.0 PL=1
CALL JOB:EXTRUDE
MOVL C00443 V=20.0 PL=1
MOVL C00444 V=130.0 PL=1
MOVL C00445 V=130.0 PL=1
CALL JOB:EXTRUDE
MOVL C00446 V=60.0 PL=1
CALL JOB:EXTRUDE
MOVL C00447 V=60.0 PL=1
CALL JOB:EXTRUDE
MOVL C00448 V=60.0 PL=1
CALL JOB:EXTRUDE
MOVL C00449 V=60.0 PL=1
MOVL C00450 V=130.0 PL=1
CALL JOB:EXTRUDE
MOVL C00451 V=30.0 PL=1
CALL JOB:EXTRUDE
MOVL C00452 V=30.0 PL=1
CALL JOB:EXTRUDE
MOVL C00453 V=30.0 PL=1
CALL JOB:EXTRUDE
MOVL C00454 V=30.0 PL=1
CALL JOB:EXTRUDE
MOVL C00455 V=30.0 PL=1
CALL JOB:EXTRUDE
MOVL C00456 V=30.0 PL=1
CALL JOB:EXTRUDE
MOVL C00457 V=30.0 PL=1
CALL JOB:EXTRUDE
MOVL C00458 V=30.0 PL=1
MOVL C00459 V=130.0 PL=1
MOVL C00460 V=130.0 PL=1
CALL JOB:EXTRUDE
MOVL C00461 V=20.0 PL=1
MOVL C00462 V=130.0 PL=1
MOVL C00463 V=130.0 PL=1
CALL JOB:EXTRUDE
MOVL C00464 V=60.0 PL=1
CALL JOB:EXTRUDE
MOVL C00465 V=60.0 PL=1
CALL JOB:EXTRUDE
MOVL C00466 V=60.0 PL=1
CALL JOB:EXTRUDE
MOVL C00467 V=60.0 PL=1
MOVL C00468 V=130.0 PL=1
CALL JOB:EXTRUDE
MOVL C00469 V=30.0 PL=1
CALL JOB:EXTRUDE
MOVL C00470 V=30.0 PL=1
CALL JOB:EXTRUDE
MOVL C00471 V=30.0 PL=1
CALL JOB:EXTRUDE
MOVL C00472 V=30.0 PL=1
CALL JOB:EXTRUDE
MOVL C00473 V=30.0 PL=1
CALL JOB:EXTRUDE
MOVL C00474 V=30.0 PL=1
CALL JOB:EXTRUDE
MOVL C00475 V=30.0 PL=1
CALL JOB:EXTRUDE
MOVL C00476 V=30.0 PL=1
MOVL C00477 V=130.0 PL=1
MOVL C00478 V=130.0 PL=1
CALL JOB:EXTRUDE
MOVL C00479 V=20.0 PL=1
MOVL C00480 V=130.0 PL=1
MOVL C00481 V=130.0 PL=1
CALL JOB:EXTRUDE
MOVL C00482 V=60.0 PL=1
CALL JOB:EXTRUDE
MOVL C00483 V=60.0 PL=1
CALL JOB:EXTRUDE
MOVL C00484 V=60.0 PL=1
CALL JOB:EXTRUDE
MOVL C00485 V=60.0 PL=1
MOVL C00486 V=130.0 PL=1
CALL JOB:EXTRUDE
MOVL C00487 V=30.0 PL=1
CALL JOB:EXTRUDE
MOVL C00488 V=30.0 PL=1
CALL JOB:EXTRUDE
MOVL C00489 V=30.0 PL=1
CALL JOB:EXTRUDE
MOVL C00490 V=30.0 PL=1
CALL JOB:EXTRUDE
MOVL C00491 V=30.0 PL=1
CALL JOB:EXTRUDE
MOVL C00492 V=30.0 PL=1
CALL JOB:EXTRUDE
MOVL C00493 V=30.0 PL=1
CALL JOB:EXTRUDE
MOVL C00494 V=30.0 PL=1
MOVL C00495 V=130.0 PL=1
MOVL C00496 V=130.0 PL=1
CALL JOB:EXTRUDE
MOVL C00497 V=20.0 PL=1
MOVL C00498 V=130.0 PL=1
MOVL C00499 V=130.0 PL=1
CALL JOB:EXTRUDE
MOVL C00500 V=60.0 PL=1
CALL JOB:EXTRUDE
MOVL C00501 V=60.0 PL=1
CALL JOB:EXTRUDE
MOVL C00502 V=60.0 PL=1
CALL JOB:EXTRUDE
MOVL C00503 V=60.0 PL=1
MOVL C00504 V=130.0 PL=1
CALL JOB:EXTRUDE
MOVL C00505 V=30.0 PL=1
CALL JOB:EXTRUDE
MOVL C00506 V=30.0 PL=1
CALL JOB:EXTRUDE
MOVL C00507 V=30.0 PL=1
CALL JOB:EXTRUDE
MOVL C00508 V=30.0 PL=1
CALL JOB:EXTRUDE
MOVL C00509 V=30.0 PL=1
CALL JOB:EXTRUDE
MOVL C00510 V=30.0 PL=1
CALL JOB:EXTRUDE
MOVL C00511 V=30.0 PL=1
CALL JOB:EXTRUDE
MOVL C00512 V=30.0 PL=1
CALL JOB:EXTRUDE
MOVL C00513 V=30.0 PL=1
CALL JOB:EXTRUDE
MOVL C00514 V=30.0 PL=1
CALL JOB:EXTRUDE
MOVL C00515 V=30.0 PL=1
CALL JOB:EXTRUDE
MOVL C00516 V=30.0 PL=1
MOVL C00517 V=130.0 PL=1
MOVL C00518 V=130.0 PL=1
CALL JOB:EXTRUDE
MOVL C00519 V=20.0 PL=1
CALL JOB:SETRPM(
CALL JOB:MCODEHA
MOVL C00520 V=130.0 PL=1
MOVL C00521 V=130.0 PL=1
CALL JOB:EXTRUDE
MOVL C00522 V=60.0 PL=1
CALL JOB:EXTRUDE
MOVL C00523 V=60.0 PL=1
CALL JOB:EXTRUDE
MOVL C00524 V=60.0 PL=1
CALL JOB:EXTRUDE
MOVL C00525 V=60.0 PL=1
MOVL C00526 V=130.0 PL=1
CALL JOB:EXTRUDE
MOVL C00527 V=30.0 PL=1
CALL JOB:EXTRUDE
MOVL C00528 V=30.0 PL=1
CALL JOB:EXTRUDE
MOVL C00529 V=30.0 PL=1
CALL JOB:EXTRUDE
MOVL C00530 V=30.0 PL=1
CALL JOB:EXTRUDE
MOVL C00531 V=30.0 PL=1
CALL JOB:EXTRUDE
MOVL C00532 V=30.0 PL=1
CALL JOB:EXTRUDE
MOVL C00533 V=30.0 PL=1
CALL JOB:EXTRUDE
MOVL C00534 V=30.0 PL=1
CALL JOB:EXTRUDE
MOVL C00535 V=30.0 PL=1
CALL JOB:EXTRUDE
MOVL C00536 V=30.0 PL=1
CALL JOB:EXTRUDE
MOVL C00537 V=30.0 PL=1
CALL JOB:EXTRUDE
MOVL C00538 V=30.0 PL=1
MOVL C00539 V=130.0 PL=1
MOVL C00540 V=130.0 PL=1
CALL JOB:EXTRUDE
MOVL C00541 V=20.0 PL=1
MOVL C00542 V=130.0 PL=1
MOVL C00543 V=130.0 PL=1
CALL JOB:EXTRUDE
MOVL C00544 V=60.0 PL=1
CALL JOB:EXTRUDE
MOVL C00545 V=60.0 PL=1
CALL JOB:EXTRUDE
MOVL C00546 V=60.0 PL=1
CALL JOB:EXTRUDE
MOVL C00547 V=60.0 PL=1
MOVL C00548 V=130.0 PL=1
CALL JOB:EXTRUDE
MOVL C00549 V=30.0 PL=1
CALL JOB:EXTRUDE
MOVL C00550 V=30.0 PL=1
CALL JOB:EXTRUDE
MOVL C00551 V=30.0 PL=1
CALL JOB:EXTRUDE
MOVL C00552 V=30.0 PL=1
CALL JOB:EXTRUDE
MOVL C00553 V=30.0 PL=1
CALL JOB:EXTRUDE
MOVL C00554 V=30.0 PL=1
CALL JOB:EXTRUDE
MOVL C00555 V=30.0 PL=1
CALL JOB:EXTRUDE
MOVL C00556 V=30.0 PL=1
CALL JOB:EXTRUDE
MOVL C00557 V=30.0 PL=1
CALL JOB:EXTRUDE
MOVL C00558 V=30.0 PL=1
CALL JOB:EXTRUDE
MOVL C00559 V=30.0 PL=1
CALL JOB:EXTRUDE
MOVL C00560 V=30.0 PL=1
MOVL C00561 V=130.0 PL=1
MOVL C00562 V=130.0 PL=1
CALL JOB:EXTRUDE
MOVL C00563 V=20.0 PL=1
MOVL C00564 V=130.0 PL=1
MOVL C00565 V=130.0 PL=1
CALL JOB:EXTRUDE
MOVL C00566 V=60.0 PL=1
CALL JOB:EXTRUDE
MOVL C00567 V=60.0 PL=1
CALL JOB:EXTRUDE
MOVL C00568 V=60.0 PL=1
CALL JOB:EXTRUDE
MOVL C00569 V=60.0 PL=1
MOVL C00570 V=130.0 PL=1
CALL JOB:EXTRUDE
MOVL C00571 V=30.0 PL=1
CALL JOB:EXTRUDE
MOVL C00572 V=30.0 PL=1
CALL JOB:EXTRUDE
MOVL C00573 V=30.0 PL=1
CALL JOB:EXTRUDE
MOVL C00574 V=30.0 PL=1
CALL JOB:EXTRUDE
MOVL C00575 V=30.0 PL=1
CALL JOB:EXTRUDE
MOVL C00576 V=30.0 PL=1
CALL JOB:EXTRUDE
MOVL C00577 V=30.0 PL=1
CALL JOB:EXTRUDE
MOVL C00578 V=30.0 PL=1
CALL JOB:EXTRUDE
MOVL C00579 V=30.0 PL=1
CALL JOB:EXTRUDE
MOVL C00580 V=30.0 PL=1
CALL JOB:EXTRUDE
MOVL C00581 V=30.0 PL=1
CALL JOB:EXTRUDE
MOVL C00582 V=30.0 PL=1
MOVL C00583 V=130.0 PL=1
MOVL C00584 V=130.0 PL=1
CALL JOB:EXTRUDE
MOVL C00585 V=20.0 PL=1
MOVL C00586 V=130.0 PL=1
MOVL C00587 V=130.0 PL=1
CALL JOB:EXTRUDE
MOVL C00588 V=60.0 PL=1
CALL JOB:EXTRUDE
MOVL C00589 V=60.0 PL=1
CALL JOB:EXTRUDE
MOVL C00590 V=60.0 PL=1
CALL JOB:EXTRUDE
MOVL C00591 V=60.0 PL=1
MOVL C00592 V=130.0 PL=1
CALL JOB:EXTRUDE
MOVL C00593 V=30.0 PL=1
CALL JOB:EXTRUDE
MOVL C00594 V=30.0 PL=1
CALL JOB:EXTRUDE
MOVL C00595 V=30.0 PL=1
CALL JOB:EXTRUDE
MOVL C00596 V=30.0 PL=1
CALL JOB:EXTRUDE
MOVL C00597 V=30.0 PL=1
CALL JOB:EXTRUDE
MOVL C00598 V=30.0 PL=1
CALL JOB:EXTRUDE
MOVL C00599 V=30.0 PL=1
CALL JOB:EXTRUDE
MOVL C00600 V=30.0 PL=1
CALL JOB:EXTRUDE
MOVL C00601 V=30.0 PL=1
CALL JOB:EXTRUDE
MOVL C00602 V=30.0 PL=1
CALL JOB:EXTRUDE
MOVL C00603 V=30.0 PL=1
CALL JOB:EXTRUDE
MOVL C00604 V=30.0 PL=1
MOVL C00605 V=130.0 PL=1
MOVL C00606 V=130.0 PL=1
CALL JOB:EXTRUDE
MOVL C00607 V=20.0 PL=1
MOVL C00608 V=130.0 PL=1
MOVL C00609 V=130.0 PL=1
CALL JOB:EXTRUDE
MOVL C00610 V=60.0 PL=1
CALL JOB:EXTRUDE
MOVL C00611 V=60.0 PL=1
CALL JOB:EXTRUDE
MOVL C00612 V=60.0 PL=1
CALL JOB:EXTRUDE
MOVL C00613 V=60.0 PL=1
MOVL C00614 V=130.0 PL=1
CALL JOB:EXTRUDE
MOVL C00615 V=30.0 PL=1
CALL JOB:EXTRUDE
MOVL C00616 V=30.0 PL=1
CALL JOB:EXTRUDE
MOVL C00617 V=30.0 PL=1
CALL JOB:EXTRUDE
MOVL C00618 V=30.0 PL=1
CALL JOB:EXTRUDE
MOVL C00619 V=30.0 PL=1
CALL JOB:EXTRUDE
MOVL C00620 V=30.0 PL=1
CALL JOB:EXTRUDE
MOVL C00621 V=30.0 PL=1
CALL JOB:EXTRUDE
MOVL C00622 V=30.0 PL=1
CALL JOB:EXTRUDE
MOVL C00623 V=30.0 PL=1
CALL JOB:EXTRUDE
MOVL C00624 V=30.0 PL=1
CALL JOB:EXTRUDE
MOVL C00625 V=30.0 PL=1
CALL JOB:EXTRUDE
MOVL C00626 V=30.0 PL=1
MOVL C00627 V=130.0 PL=1
MOVL C00628 V=130.0 PL=1
CALL JOB:EXTRUDE
MOVL C00629 V=20.0 PL=1
MOVL C00630 V=130.0 PL=1
MOVL C00631 V=130.0 PL=1
CALL JOB:EXTRUDE
MOVL C00632 V=60.0 PL=1
CALL JOB:EXTRUDE
MOVL C00633 V=60.0 PL=1
CALL JOB:EXTRUDE
MOVL C00634 V=60.0 PL=1
CALL JOB:EXTRUDE
MOVL C00635 V=60.0 PL=1
MOVL C00636 V=130.0 PL=1
CALL JOB:EXTRUDE
MOVL C00637 V=30.0 PL=1
CALL JOB:EXTRUDE
MOVL C00638 V=30.0 PL=1
CALL JOB:EXTRUDE
MOVL C00639 V=30.0 PL=1
CALL JOB:EXTRUDE
MOVL C00640 V=30.0 PL=1
CALL JOB:EXTRUDE
MOVL C00641 V=30.0 PL=1
CALL JOB:EXTRUDE
MOVL C00642 V=30.0 PL=1
CALL JOB:EXTRUDE
MOVL C00643 V=30.0 PL=1
CALL JOB:EXTRUDE
MOVL C00644 V=30.0 PL=1
CALL JOB:EXTRUDE
MOVL C00645 V=30.0 PL=1
CALL JOB:EXTRUDE
MOVL C00646 V=30.0 PL=1
CALL JOB:EXTRUDE
MOVL C00647 V=30.0 PL=1
CALL JOB:EXTRUDE
MOVL C00648 V=30.0 PL=1
MOVL C00649 V=130.0 PL=1
MOVL C00650 V=130.0 PL=1
CALL JOB:EXTRUDE
MOVL C00651 V=20.0 PL=1
MOVL C00652 V=130.0 PL=1
MOVL C00653 V=130.0 PL=1
CALL JOB:EXTRUDE
MOVL C00654 V=60.0 PL=1
CALL JOB:EXTRUDE
MOVL C00655 V=60.0 PL=1
CALL JOB:EXTRUDE
MOVL C00656 V=60.0 PL=1
CALL JOB:EXTRUDE
MOVL C00657 V=60.0 PL=1
MOVL C00658 V=130.0 PL=1
CALL JOB:EXTRUDE
MOVL C00659 V=30.0 PL=1
CALL JOB:EXTRUDE
MOVL C00660 V=30.0 PL=1
CALL JOB:EXTRUDE
MOVL C00661 V=30.0 PL=1
CALL JOB:EXTRUDE
MOVL C00662 V=30.0 PL=1
CALL JOB:EXTRUDE
MOVL C00663 V=30.0 PL=1
CALL JOB:EXTRUDE
MOVL C00664 V=30.0 PL=1
CALL JOB:EXTRUDE
MOVL C00665 V=30.0 PL=1
CALL JOB:EXTRUDE
MOVL C00666 V=30.0 PL=1
CALL JOB:EXTRUDE
MOVL C00667 V=30.0 PL=1
CALL JOB:EXTRUDE
MOVL C00668 V=30.0 PL=1
CALL JOB:EXTRUDE
MOVL C00669 V=30.0 PL=1
CALL JOB:EXTRUDE
MOVL C00670 V=30.0 PL=1
MOVL C00671 V=130.0 PL=1
MOVL C00672 V=130.0 PL=1
CALL JOB:EXTRUDE
MOVL C00673 V=20.0 PL=1
MOVL C00674 V=130.0 PL=1
MOVL C00675 V=130.0 PL=1
CALL JOB:EXTRUDE
MOVL C00676 V=60.0 PL=1
CALL JOB:EXTRUDE
MOVL C00677 V=60.0 PL=1
CALL JOB:EXTRUDE
MOVL C00678 V=60.0 PL=1
CALL JOB:EXTRUDE
MOVL C00679 V=60.0 PL=1
MOVL C00680 V=130.0 PL=1
CALL JOB:EXTRUDE
MOVL C00681 V=30.0 PL=1
CALL JOB:EXTRUDE
MOVL C00682 V=30.0 PL=1
CALL JOB:EXTRUDE
MOVL C00683 V=30.0 PL=1
CALL JOB:EXTRUDE
MOVL C00684 V=30.0 PL=1
CALL JOB:EXTRUDE
MOVL C00685 V=30.0 PL=1
CALL JOB:EXTRUDE
MOVL C00686 V=30.0 PL=1
CALL JOB:EXTRUDE
MOVL C00687 V=30.0 PL=1
CALL JOB:EXTRUDE
MOVL C00688 V=30.0 PL=1
CALL JOB:EXTRUDE
MOVL C00689 V=30.0 PL=1
CALL JOB:EXTRUDE
MOVL C00690 V=30.0 PL=1
CALL JOB:EXTRUDE
MOVL C00691 V=30.0 PL=1
CALL JOB:EXTRUDE
MOVL C00692 V=30.0 PL=1
MOVL C00693 V=130.0 PL=1
MOVL C00694 V=130.0 PL=1
CALL JOB:EXTRUDE
MOVL C00695 V=20.0 PL=1
MOVL C00696 V=130.0 PL=1
MOVL C00697 V=130.0 PL=1
CALL JOB:EXTRUDE
MOVL C00698 V=60.0 PL=1
CALL JOB:EXTRUDE
MOVL C00699 V=60.0 PL=1
CALL JOB:EXTRUDE
MOVL C00700 V=60.0 PL=1
CALL JOB:EXTRUDE
MOVL C00701 V=60.0 PL=1
MOVL C00702 V=130.0 PL=1
CALL JOB:EXTRUDE
MOVL C00703 V=30.0 PL=1
CALL JOB:EXTRUDE
MOVL C00704 V=30.0 PL=1
CALL JOB:EXTRUDE
MOVL C00705 V=30.0 PL=1
CALL JOB:EXTRUDE
MOVL C00706 V=30.0 PL=1
CALL JOB:EXTRUDE
MOVL C00707 V=30.0 PL=1
CALL JOB:EXTRUDE
MOVL C00708 V=30.0 PL=1
CALL JOB:EXTRUDE
MOVL C00709 V=30.0 PL=1
CALL JOB:EXTRUDE
MOVL C00710 V=30.0 PL=1
CALL JOB:EXTRUDE
MOVL C00711 V=30.0 PL=1
CALL JOB:EXTRUDE
MOVL C00712 V=30.0 PL=1
CALL JOB:EXTRUDE
MOVL C00713 V=30.0 PL=1
CALL JOB:EXTRUDE
MOVL C00714 V=30.0 PL=1
MOVL C00715 V=130.0 PL=1
MOVL C00716 V=130.0 PL=1
CALL JOB:EXTRUDE
MOVL C00717 V=20.0 PL=1
MOVL C00718 V=130.0 PL=1
MOVL C00719 V=130.0 PL=1
CALL JOB:EXTRUDE
MOVL C00720 V=60.0 PL=1
CALL JOB:EXTRUDE
MOVL C00721 V=60.0 PL=1
CALL JOB:EXTRUDE
MOVL C00722 V=60.0 PL=1
CALL JOB:EXTRUDE
MOVL C00723 V=60.0 PL=1
MOVL C00724 V=130.0 PL=1
CALL JOB:EXTRUDE
MOVL C00725 V=30.0 PL=1
CALL JOB:EXTRUDE
MOVL C00726 V=30.0 PL=1
CALL JOB:EXTRUDE
MOVL C00727 V=30.0 PL=1
CALL JOB:EXTRUDE
MOVL C00728 V=30.0 PL=1
CALL JOB:EXTRUDE
MOVL C00729 V=30.0 PL=1
CALL JOB:EXTRUDE
MOVL C00730 V=30.0 PL=1
CALL JOB:EXTRUDE
MOVL C00731 V=30.0 PL=1
CALL JOB:EXTRUDE
MOVL C00732 V=30.0 PL=1
CALL JOB:EXTRUDE
MOVL C00733 V=30.0 PL=1
CALL JOB:EXTRUDE
MOVL C00734 V=30.0 PL=1
CALL JOB:EXTRUDE
MOVL C00735 V=30.0 PL=1
CALL JOB:EXTRUDE
MOVL C00736 V=30.0 PL=1
MOVL C00737 V=130.0 PL=1
MOVL C00738 V=130.0 PL=1
CALL JOB:EXTRUDE
MOVL C00739 V=20.0 PL=1
MOVL C00740 V=130.0 PL=1
MOVL C00741 V=130.0 PL=1
CALL JOB:EXTRUDE
MOVL C00742 V=60.0 PL=1
CALL JOB:EXTRUDE
MOVL C00743 V=60.0 PL=1
CALL JOB:EXTRUDE
MOVL C00744 V=60.0 PL=1
CALL JOB:EXTRUDE
MOVL C00745 V=60.0 PL=1
MOVL C00746 V=130.0 PL=1
CALL JOB:EXTRUDE
MOVL C00747 V=30.0 PL=1
CALL JOB:EXTRUDE
MOVL C00748 V=30.0 PL=1
CALL JOB:EXTRUDE
MOVL C00749 V=30.0 PL=1
CALL JOB:EXTRUDE
MOVL C00750 V=30.0 PL=1
CALL JOB:EXTRUDE
MOVL C00751 V=30.0 PL=1
CALL JOB:EXTRUDE
MOVL C00752 V=30.0 PL=1
CALL JOB:EXTRUDE
MOVL C00753 V=30.0 PL=1
CALL JOB:EXTRUDE
MOVL C00754 V=30.0 PL=1
CALL JOB:EXTRUDE
MOVL C00755 V=30.0 PL=1
CALL JOB:EXTRUDE
MOVL C00756 V=30.0 PL=1
CALL JOB:EXTRUDE
MOVL C00757 V=30.0 PL=1
CALL JOB:EXTRUDE
MOVL C00758 V=30.0 PL=1
MOVL C00759 V=130.0 PL=1
MOVL C00760 V=130.0 PL=1
CALL JOB:EXTRUDE
MOVL C00761 V=20.0 PL=1
MOVL C00762 V=130.0 PL=1
MOVL C00763 V=130.0 PL=1
CALL JOB:EXTRUDE
MOVL C00764 V=60.0 PL=1
CALL JOB:EXTRUDE
MOVL C00765 V=60.0 PL=1
CALL JOB:EXTRUDE
MOVL C00766 V=60.0 PL=1
CALL JOB:EXTRUDE
MOVL C00767 V=60.0 PL=1
MOVL C00768 V=130.0 PL=1
CALL JOB:EXTRUDE
MOVL C00769 V=30.0 PL=1
CALL JOB:EXTRUDE
MOVL C00770 V=30.0 PL=1
CALL JOB:EXTRUDE
MOVL C00771 V=30.0 PL=1
CALL JOB:EXTRUDE
MOVL C00772 V=30.0 PL=1
CALL JOB:EXTRUDE
MOVL C00773 V=30.0 PL=1
CALL JOB:EXTRUDE
MOVL C00774 V=30.0 PL=1
CALL JOB:EXTRUDE
MOVL C00775 V=30.0 PL=1
CALL JOB:EXTRUDE
MOVL C00776 V=30.0 PL=1
CALL JOB:EXTRUDE
MOVL C00777 V=30.0 PL=1
CALL JOB:EXTRUDE
MOVL C00778 V=30.0 PL=1
CALL JOB:EXTRUDE
MOVL C00779 V=30.0 PL=1
CALL JOB:EXTRUDE
MOVL C00780 V=30.0 PL=1
MOVL C00781 V=130.0 PL=1
MOVL C00782 V=130.0 PL=1
CALL JOB:EXTRUDE
MOVL C00783 V=20.0 PL=1
MOVL C00784 V=130.0 PL=1
MOVL C00785 V=130.0 PL=1
CALL JOB:EXTRUDE
MOVL C00786 V=60.0 PL=1
CALL JOB:EXTRUDE
MOVL C00787 V=60.0 PL=1
CALL JOB:EXTRUDE
MOVL C00788 V=60.0 PL=1
CALL JOB:EXTRUDE
MOVL C00789 V=60.0 PL=1
MOVL C00790 V=130.0 PL=1
CALL JOB:EXTRUDE
MOVL C00791 V=30.0 PL=1
CALL JOB:EXTRUDE
MOVL C00792 V=30.0 PL=1
CALL JOB:EXTRUDE
MOVL C00793 V=30.0 PL=1
CALL JOB:EXTRUDE
MOVL C00794 V=30.0 PL=1
CALL JOB:EXTRUDE
MOVL C00795 V=30.0 PL=1
CALL JOB:EXTRUDE
MOVL C00796 V=30.0 PL=1
CALL JOB:EXTRUDE
MOVL C00797 V=30.0 PL=1
CALL JOB:EXTRUDE
MOVL C00798 V=30.0 PL=1
CALL JOB:EXTRUDE
MOVL C00799 V=30.0 PL=1
CALL JOB:EXTRUDE
MOVL C00800 V=30.0 PL=1
CALL JOB:EXTRUDE
MOVL C00801 V=30.0 PL=1
CALL JOB:EXTRUDE
MOVL C00802 V=30.0 PL=1
MOVL C00803 V=130.0 PL=1
MOVL C00804 V=130.0 PL=1
CALL JOB:EXTRUDE
MOVL C00805 V=20.0 PL=1
MOVL C00806 V=130.0 PL=1
MOVL C00807 V=130.0 PL=1
CALL JOB:EXTRUDE
MOVL C00808 V=60.0 PL=1
CALL JOB:EXTRUDE
MOVL C00809 V=60.0 PL=1
CALL JOB:EXTRUDE
MOVL C00810 V=60.0 PL=1
CALL JOB:EXTRUDE
MOVL C00811 V=60.0 PL=1
MOVL C00812 V=130.0 PL=1
CALL JOB:EXTRUDE
MOVL C00813 V=30.0 PL=1
CALL JOB:EXTRUDE
MOVL C00814 V=30.0 PL=1
CALL JOB:EXTRUDE
MOVL C00815 V=30.0 PL=1
CALL JOB:EXTRUDE
MOVL C00816 V=30.0 PL=1
CALL JOB:EXTRUDE
MOVL C00817 V=30.0 PL=1
CALL JOB:EXTRUDE
MOVL C00818 V=30.0 PL=1
CALL JOB:EXTRUDE
MOVL C00819 V=30.0 PL=1
CALL JOB:EXTRUDE
MOVL C00820 V=30.0 PL=1
CALL JOB:EXTRUDE
MOVL C00821 V=30.0 PL=1
CALL JOB:EXTRUDE
MOVL C00822 V=30.0 PL=1
CALL JOB:EXTRUDE
MOVL C00823 V=30.0 PL=1
CALL JOB:EXTRUDE
MOVL C00824 V=30.0 PL=1
MOVL C00825 V=130.0 PL=1
MOVL C00826 V=130.0 PL=1
CALL JOB:EXTRUDE
MOVL C00827 V=20.0 PL=1
MOVL C00828 V=130.0 PL=1
MOVL C00829 V=130.0 PL=1
CALL JOB:EXTRUDE
MOVL C00830 V=60.0 PL=1
CALL JOB:EXTRUDE
MOVL C00831 V=60.0 PL=1
CALL JOB:EXTRUDE
MOVL C00832 V=60.0 PL=1
CALL JOB:EXTRUDE
MOVL C00833 V=60.0 PL=1
MOVL C00834 V=130.0 PL=1
CALL JOB:EXTRUDE
MOVL C00835 V=30.0 PL=1
CALL JOB:EXTRUDE
MOVL C00836 V=30.0 PL=1
CALL JOB:EXTRUDE
MOVL C00837 V=30.0 PL=1
CALL JOB:EXTRUDE
MOVL C00838 V=30.0 PL=1
CALL JOB:EXTRUDE
MOVL C00839 V=30.0 PL=1
CALL JOB:EXTRUDE
MOVL C00840 V=30.0 PL=1
CALL JOB:EXTRUDE
MOVL C00841 V=30.0 PL=1
CALL JOB:EXTRUDE
MOVL C00842 V=30.0 PL=1
CALL JOB:EXTRUDE
MOVL C00843 V=30.0 PL=1
CALL JOB:EXTRUDE
MOVL C00844 V=30.0 PL=1
CALL JOB:EXTRUDE
MOVL C00845 V=30.0 PL=1
CALL JOB:EXTRUDE
MOVL C00846 V=30.0 PL=1
MOVL C00847 V=130.0 PL=1
MOVL C00848 V=130.0 PL=1
CALL JOB:EXTRUDE
MOVL C00849 V=20.0 PL=1
MOVL C00850 V=130.0 PL=1
MOVL C00851 V=130.0 PL=1
CALL JOB:EXTRUDE
MOVL C00852 V=60.0 PL=1
CALL JOB:EXTRUDE
MOVL C00853 V=60.0 PL=1
CALL JOB:EXTRUDE
MOVL C00854 V=60.0 PL=1
CALL JOB:EXTRUDE
MOVL C00855 V=60.0 PL=1
MOVL C00856 V=130.0 PL=1
CALL JOB:EXTRUDE
MOVL C00857 V=30.0 PL=1
CALL JOB:EXTRUDE
MOVL C00858 V=30.0 PL=1
CALL JOB:EXTRUDE
MOVL C00859 V=30.0 PL=1
CALL JOB:EXTRUDE
MOVL C00860 V=30.0 PL=1
CALL JOB:EXTRUDE
MOVL C00861 V=30.0 PL=1
CALL JOB:EXTRUDE
MOVL C00862 V=30.0 PL=1
CALL JOB:EXTRUDE
MOVL C00863 V=30.0 PL=1
CALL JOB:EXTRUDE
MOVL C00864 V=30.0 PL=1
CALL JOB:EXTRUDE
MOVL C00865 V=30.0 PL=1
CALL JOB:EXTRUDE
MOVL C00866 V=30.0 PL=1
CALL JOB:EXTRUDE
MOVL C00867 V=30.0 PL=1
CALL JOB:EXTRUDE
MOVL C00868 V=30.0 PL=1
MOVL C00869 V=130.0 PL=1
MOVL C00870 V=130.0 PL=1
CALL JOB:EXTRUDE
MOVL C00871 V=20.0 PL=1
MOVL C00872 V=130.0 PL=1
MOVL C00873 V=130.0 PL=1
CALL JOB:EXTRUDE
MOVL C00874 V=60.0 PL=1
CALL JOB:EXTRUDE
MOVL C00875 V=60.0 PL=1
CALL JOB:EXTRUDE
MOVL C00876 V=60.0 PL=1
CALL JOB:EXTRUDE
MOVL C00877 V=60.0 PL=1
MOVL C00878 V=130.0 PL=1
CALL JOB:EXTRUDE
MOVL C00879 V=30.0 PL=1
CALL JOB:EXTRUDE
MOVL C00880 V=30.0 PL=1
CALL JOB:EXTRUDE
MOVL C00881 V=30.0 PL=1
CALL JOB:EXTRUDE
MOVL C00882 V=30.0 PL=1
CALL JOB:EXTRUDE
MOVL C00883 V=30.0 PL=1
CALL JOB:EXTRUDE
MOVL C00884 V=30.0 PL=1
CALL JOB:EXTRUDE
MOVL C00885 V=30.0 PL=1
CALL JOB:EXTRUDE
MOVL C00886 V=30.0 PL=1
CALL JOB:EXTRUDE
MOVL C00887 V=30.0 PL=1
CALL JOB:EXTRUDE
MOVL C00888 V=30.0 PL=1
CALL JOB:EXTRUDE
MOVL C00889 V=30.0 PL=1
CALL JOB:EXTRUDE
MOVL C00890 V=30.0 PL=1
MOVL C00891 V=130.0 PL=1
MOVL C00892 V=130.0 PL=1
CALL JOB:EXTRUDE
MOVL C00893 V=20.0 PL=1
MOVL C00894 V=130.0 PL=1
MOVL C00895 V=130.0 PL=1
CALL JOB:EXTRUDE
MOVL C00896 V=60.0 PL=1
CALL JOB:EXTRUDE
MOVL C00897 V=60.0 PL=1
CALL JOB:EXTRUDE
MOVL C00898 V=60.0 PL=1
CALL JOB:EXTRUDE
MOVL C00899 V=60.0 PL=1
MOVL C00900 V=130.0 PL=1
CALL JOB:EXTRUDE
MOVL C00901 V=30.0 PL=1
CALL JOB:EXTRUDE
MOVL C00902 V=30.0 PL=1
CALL JOB:EXTRUDE
MOVL C00903 V=30.0 PL=1
CALL JOB:EXTRUDE
MOVL C00904 V=30.0 PL=1
CALL JOB:EXTRUDE
MOVL C00905 V=30.0 PL=1
CALL JOB:EXTRUDE
MOVL C00906 V=30.0 PL=1
CALL JOB:EXTRUDE
MOVL C00907 V=30.0 PL=1
CALL JOB:EXTRUDE
MOVL C00908 V=30.0 PL=1
CALL JOB:EXTRUDE
MOVL C00909 V=30.0 PL=1
CALL JOB:EXTRUDE
MOVL C00910 V=30.0 PL=1
CALL JOB:EXTRUDE
MOVL C00911 V=30.0 PL=1
CALL JOB:EXTRUDE
MOVL C00912 V=30.0 PL=1
MOVL C00913 V=130.0 PL=1
MOVL C00914 V=130.0 PL=1
CALL JOB:EXTRUDE
MOVL C00915 V=20.0 PL=1
MOVL C00916 V=130.0 PL=1
MOVL C00917 V=130.0 PL=1
CALL JOB:EXTRUDE
MOVL C00918 V=60.0 PL=1
CALL JOB:EXTRUDE
MOVL C00919 V=60.0 PL=1
CALL JOB:EXTRUDE
MOVL C00920 V=60.0 PL=1
CALL JOB:EXTRUDE
MOVL C00921 V=60.0 PL=1
MOVL C00922 V=130.0 PL=1
CALL JOB:EXTRUDE
MOVL C00923 V=30.0 PL=1
CALL JOB:EXTRUDE
MOVL C00924 V=30.0 PL=1
CALL JOB:EXTRUDE
MOVL C00925 V=30.0 PL=1
CALL JOB:EXTRUDE
MOVL C00926 V=30.0 PL=1
CALL JOB:EXTRUDE
MOVL C00927 V=30.0 PL=1
CALL JOB:EXTRUDE
MOVL C00928 V=30.0 PL=1
CALL JOB:EXTRUDE
MOVL C00929 V=30.0 PL=1
CALL JOB:EXTRUDE
MOVL C00930 V=30.0 PL=1
CALL JOB:EXTRUDE
MOVL C00931 V=30.0 PL=1
CALL JOB:EXTRUDE
MOVL C00932 V=30.0 PL=1
CALL JOB:EXTRUDE
MOVL C00933 V=30.0 PL=1
CALL JOB:EXTRUDE
MOVL C00934 V=30.0 PL=1
MOVL C00935 V=130.0 PL=1
MOVL C00936 V=130.0 PL=1
CALL JOB:EXTRUDE
MOVL C00937 V=20.0 PL=1
MOVL C00938 V=130.0 PL=1
MOVL C00939 V=130.0 PL=1
CALL JOB:EXTRUDE
MOVL C00940 V=60.0 PL=1
CALL JOB:EXTRUDE
MOVL C00941 V=60.0 PL=1
CALL JOB:EXTRUDE
MOVL C00942 V=60.0 PL=1
CALL JOB:EXTRUDE
MOVL C00943 V=60.0 PL=1
MOVL C00944 V=130.0 PL=1
CALL JOB:EXTRUDE
MOVL C00945 V=30.0 PL=1
CALL JOB:EXTRUDE
MOVL C00946 V=30.0 PL=1
CALL JOB:EXTRUDE
MOVL C00947 V=30.0 PL=1
CALL JOB:EXTRUDE
MOVL C00948 V=30.0 PL=1
CALL JOB:EXTRUDE
MOVL C00949 V=30.0 PL=1
CALL JOB:EXTRUDE
MOVL C00950 V=30.0 PL=1
CALL JOB:EXTRUDE
MOVL C00951 V=30.0 PL=1
CALL JOB:EXTRUDE
MOVL C00952 V=30.0 PL=1
CALL JOB:EXTRUDE
MOVL C00953 V=30.0 PL=1
CALL JOB:EXTRUDE
MOVL C00954 V=30.0 PL=1
CALL JOB:EXTRUDE
MOVL C00955 V=30.0 PL=1
CALL JOB:EXTRUDE
MOVL C00956 V=30.0 PL=1
MOVL C00957 V=130.0 PL=1
MOVL C00958 V=130.0 PL=1
CALL JOB:EXTRUDE
MOVL C00959 V=20.0 PL=1
MOVL C00960 V=130.0 PL=1
MOVL C00961 V=130.0 PL=1
CALL JOB:EXTRUDE
MOVL C00962 V=60.0 PL=1
CALL JOB:EXTRUDE
MOVL C00963 V=60.0 PL=1
CALL JOB:EXTRUDE
MOVL C00964 V=60.0 PL=1
CALL JOB:EXTRUDE
MOVL C00965 V=60.0 PL=1
MOVL C00966 V=130.0 PL=1
CALL JOB:EXTRUDE
MOVL C00967 V=30.0 PL=1
CALL JOB:EXTRUDE
MOVL C00968 V=30.0 PL=1
CALL JOB:EXTRUDE
MOVL C00969 V=30.0 PL=1
CALL JOB:EXTRUDE
MOVL C00970 V=30.0 PL=1
CALL JOB:EXTRUDE
MOVL C00971 V=30.0 PL=1
CALL JOB:EXTRUDE
MOVL C00972 V=30.0 PL=1
CALL JOB:EXTRUDE
MOVL C00973 V=30.0 PL=1
CALL JOB:EXTRUDE
MOVL C00974 V=30.0 PL=1
CALL JOB:EXTRUDE
MOVL C00975 V=30.0 PL=1
CALL JOB:EXTRUDE
MOVL C00976 V=30.0 PL=1
CALL JOB:EXTRUDE
MOVL C00977 V=30.0 PL=1
CALL JOB:EXTRUDE
MOVL C00978 V=30.0 PL=1
MOVL C00979 V=130.0 PL=1
MOVL C00980 V=130.0 PL=1
CALL JOB:EXTRUDE
MOVL C00981 V=20.0 PL=1
CALL JOB:SETRPM(
CALL JOB:MCODEHA
MOVL C00982 V=130.0 PL=1
MOVL C00983 V=130.0 PL=1
CALL JOB:EXTRUDE
MOVL C00984 V=60.0 PL=1
CALL JOB:EXTRUDE
MOVL C00985 V=60.0 PL=1
CALL JOB:EXTRUDE
MOVL C00986 V=60.0 PL=1
CALL JOB:EXTRUDE
MOVL C00987 V=60.0 PL=1
CALL JOB:EXTRUDE
MOVL C00988 V=60.0 PL=1
CALL JOB:EXTRUDE
MOVL C00989 V=60.0 PL=1
MOVL C00990 V=130.0 PL=1
CALL JOB:EXTRUDE
MOVL C00991 V=30.0 PL=1
CALL JOB:EXTRUDE
MOVL C00992 V=30.0 PL=1
CALL JOB:EXTRUDE
MOVL C00993 V=30.0 PL=1
CALL JOB:EXTRUDE
MOVL C00994 V=30.0 PL=1
CALL JOB:EXTRUDE
MOVL C00995 V=30.0 PL=1
CALL JOB:EXTRUDE
MOVL C00996 V=30.0 PL=1
CALL JOB:EXTRUDE
MOVL C00997 V=30.0 PL=1
CALL JOB:EXTRUDE
MOVL C00998 V=30.0 PL=1
CALL JOB:EXTRUDE
MOVL C00999 V=30.0 PL=1
CALL JOB:EXTRUDE
MOVL C01000 V=30.0 PL=1
CALL JOB:EXTRUDE
MOVL C01001 V=30.0 PL=1
CALL JOB:EXTRUDE
MOVL C01002 V=30.0 PL=1
MOVL C01003 V=130.0 PL=1
MOVL C01004 V=130.0 PL=1
CALL JOB:EXTRUDE
MOVL C01005 V=20.0 PL=1
MOVL C01006 V=130.0 PL=1
MOVL C01007 V=130.0 PL=1
CALL JOB:EXTRUDE
MOVL C01008 V=60.0 PL=1
CALL JOB:EXTRUDE
MOVL C01009 V=60.0 PL=1
CALL JOB:EXTRUDE
MOVL C01010 V=60.0 PL=1
CALL JOB:EXTRUDE
MOVL C01011 V=60.0 PL=1
CALL JOB:EXTRUDE
MOVL C01012 V=60.0 PL=1
CALL JOB:EXTRUDE
MOVL C01013 V=60.0 PL=1
MOVL C01014 V=130.0 PL=1
CALL JOB:EXTRUDE
MOVL C01015 V=30.0 PL=1
CALL JOB:EXTRUDE
MOVL C01016 V=30.0 PL=1
CALL JOB:EXTRUDE
MOVL C01017 V=30.0 PL=1
CALL JOB:EXTRUDE
MOVL C01018 V=30.0 PL=1
CALL JOB:EXTRUDE
MOVL C01019 V=30.0 PL=1
CALL JOB:EXTRUDE
MOVL C01020 V=30.0 PL=1
CALL JOB:EXTRUDE
MOVL C01021 V=30.0 PL=1
CALL JOB:EXTRUDE
MOVL C01022 V=30.0 PL=1
CALL JOB:EXTRUDE
MOVL C01023 V=30.0 PL=1
CALL JOB:EXTRUDE
MOVL C01024 V=30.0 PL=1
CALL JOB:EXTRUDE
MOVL C01025 V=30.0 PL=1
CALL JOB:EXTRUDE
MOVL C01026 V=30.0 PL=1
MOVL C01027 V=130.0 PL=1
MOVL C01028 V=130.0 PL=1
CALL JOB:EXTRUDE
MOVL C01029 V=20.0 PL=1
MOVL C01030 V=130.0 PL=1
MOVL C01031 V=130.0 PL=1
CALL JOB:EXTRUDE
MOVL C01032 V=60.0 PL=1
CALL JOB:EXTRUDE
MOVL C01033 V=60.0 PL=1
CALL JOB:EXTRUDE
MOVL C01034 V=60.0 PL=1
CALL JOB:EXTRUDE
MOVL C01035 V=60.0 PL=1
CALL JOB:EXTRUDE
MOVL C01036 V=60.0 PL=1
CALL JOB:EXTRUDE
MOVL C01037 V=60.0 PL=1
MOVL C01038 V=130.0 PL=1
CALL JOB:EXTRUDE
MOVL C01039 V=30.0 PL=1
CALL JOB:EXTRUDE
MOVL C01040 V=30.0 PL=1
CALL JOB:EXTRUDE
MOVL C01041 V=30.0 PL=1
CALL JOB:EXTRUDE
MOVL C01042 V=30.0 PL=1
CALL JOB:EXTRUDE
MOVL C01043 V=30.0 PL=1
CALL JOB:EXTRUDE
MOVL C01044 V=30.0 PL=1
CALL JOB:EXTRUDE
MOVL C01045 V=30.0 PL=1
CALL JOB:EXTRUDE
MOVL C01046 V=30.0 PL=1
CALL JOB:EXTRUDE
MOVL C01047 V=30.0 PL=1
CALL JOB:EXTRUDE
MOVL C01048 V=30.0 PL=1
CALL JOB:EXTRUDE
MOVL C01049 V=30.0 PL=1
CALL JOB:EXTRUDE
MOVL C01050 V=30.0 PL=1
MOVL C01051 V=130.0 PL=1
MOVL C01052 V=130.0 PL=1
CALL JOB:EXTRUDE
MOVL C01053 V=20.0 PL=1
MOVL C01054 V=130.0 PL=1
MOVL C01055 V=130.0 PL=1
CALL JOB:EXTRUDE
MOVL C01056 V=60.0 PL=1
CALL JOB:EXTRUDE
MOVL C01057 V=60.0 PL=1
CALL JOB:EXTRUDE
MOVL C01058 V=60.0 PL=1
CALL JOB:EXTRUDE
MOVL C01059 V=60.0 PL=1
CALL JOB:EXTRUDE
MOVL C01060 V=60.0 PL=1
CALL JOB:EXTRUDE
MOVL C01061 V=60.0 PL=1
MOVL C01062 V=130.0 PL=1
CALL JOB:EXTRUDE
MOVL C01063 V=30.0 PL=1
CALL JOB:EXTRUDE
MOVL C01064 V=30.0 PL=1
CALL JOB:EXTRUDE
MOVL C01065 V=30.0 PL=1
CALL JOB:EXTRUDE
MOVL C01066 V=30.0 PL=1
CALL JOB:EXTRUDE
MOVL C01067 V=30.0 PL=1
CALL JOB:EXTRUDE
MOVL C01068 V=30.0 PL=1
CALL JOB:EXTRUDE
MOVL C01069 V=30.0 PL=1
CALL JOB:EXTRUDE
MOVL C01070 V=30.0 PL=1
CALL JOB:EXTRUDE
MOVL C01071 V=30.0 PL=1
CALL JOB:EXTRUDE
MOVL C01072 V=30.0 PL=1
CALL JOB:EXTRUDE
MOVL C01073 V=30.0 PL=1
CALL JOB:EXTRUDE
MOVL C01074 V=30.0 PL=1
MOVL C01075 V=130.0 PL=1
MOVL C01076 V=130.0 PL=1
CALL JOB:EXTRUDE
MOVL C01077 V=20.0 PL=1
MOVL C01078 V=130.0 PL=1
MOVL C01079 V=130.0 PL=1
CALL JOB:EXTRUDE
MOVL C01080 V=60.0 PL=1
CALL JOB:EXTRUDE
MOVL C01081 V=60.0 PL=1
CALL JOB:EXTRUDE
MOVL C01082 V=60.0 PL=1
CALL JOB:EXTRUDE
MOVL C01083 V=60.0 PL=1
CALL JOB:EXTRUDE
MOVL C01084 V=60.0 PL=1
CALL JOB:EXTRUDE
MOVL C01085 V=60.0 PL=1
MOVL C01086 V=130.0 PL=1
CALL JOB:EXTRUDE
MOVL C01087 V=30.0 PL=1
CALL JOB:EXTRUDE
MOVL C01088 V=30.0 PL=1
CALL JOB:EXTRUDE
MOVL C01089 V=30.0 PL=1
CALL JOB:EXTRUDE
MOVL C01090 V=30.0 PL=1
CALL JOB:EXTRUDE
MOVL C01091 V=30.0 PL=1
CALL JOB:EXTRUDE
MOVL C01092 V=30.0 PL=1
CALL JOB:EXTRUDE
MOVL C01093 V=30.0 PL=1
CALL JOB:EXTRUDE
MOVL C01094 V=30.0 PL=1
CALL JOB:EXTRUDE
MOVL C01095 V=30.0 PL=1
CALL JOB:EXTRUDE
MOVL C01096 V=30.0 PL=1
CALL JOB:EXTRUDE
MOVL C01097 V=30.0 PL=1
CALL JOB:EXTRUDE
MOVL C01098 V=30.0 PL=1
MOVL C01099 V=130.0 PL=1
MOVL C01100 V=130.0 PL=1
CALL JOB:EXTRUDE
MOVL C01101 V=20.0 PL=1
MOVL C01102 V=130.0 PL=1
MOVL C01103 V=130.0 PL=1
CALL JOB:EXTRUDE
MOVL C01104 V=60.0 PL=1
CALL JOB:EXTRUDE
MOVL C01105 V=60.0 PL=1
CALL JOB:EXTRUDE
MOVL C01106 V=60.0 PL=1
CALL JOB:EXTRUDE
MOVL C01107 V=60.0 PL=1
CALL JOB:EXTRUDE
MOVL C01108 V=60.0 PL=1
CALL JOB:EXTRUDE
MOVL C01109 V=60.0 PL=1
MOVL C01110 V=130.0 PL=1
CALL JOB:EXTRUDE
MOVL C01111 V=30.0 PL=1
CALL JOB:EXTRUDE
MOVL C01112 V=30.0 PL=1
CALL JOB:EXTRUDE
MOVL C01113 V=30.0 PL=1
CALL JOB:EXTRUDE
MOVL C01114 V=30.0 PL=1
CALL JOB:EXTRUDE
MOVL C01115 V=30.0 PL=1
CALL JOB:EXTRUDE
MOVL C01116 V=30.0 PL=1
CALL JOB:EXTRUDE
MOVL C01117 V=30.0 PL=1
CALL JOB:EXTRUDE
MOVL C01118 V=30.0 PL=1
CALL JOB:EXTRUDE
MOVL C01119 V=30.0 PL=1
CALL JOB:EXTRUDE
MOVL C01120 V=30.0 PL=1
CALL JOB:EXTRUDE
MOVL C01121 V=30.0 PL=1
CALL JOB:EXTRUDE
MOVL C01122 V=30.0 PL=1
MOVL C01123 V=130.0 PL=1
MOVL C01124 V=130.0 PL=1
CALL JOB:EXTRUDE
MOVL C01125 V=20.0 PL=1
MOVL C01126 V=130.0 PL=1
MOVL C01127 V=130.0 PL=1
CALL JOB:EXTRUDE
MOVL C01128 V=60.0 PL=1
CALL JOB:EXTRUDE
MOVL C01129 V=60.0 PL=1
CALL JOB:EXTRUDE
MOVL C01130 V=60.0 PL=1
CALL JOB:EXTRUDE
MOVL C01131 V=60.0 PL=1
CALL JOB:EXTRUDE
MOVL C01132 V=60.0 PL=1
CALL JOB:EXTRUDE
MOVL C01133 V=60.0 PL=1
MOVL C01134 V=130.0 PL=1
CALL JOB:EXTRUDE
MOVL C01135 V=30.0 PL=1
CALL JOB:EXTRUDE
MOVL C01136 V=30.0 PL=1
CALL JOB:EXTRUDE
MOVL C01137 V=30.0 PL=1
CALL JOB:EXTRUDE
END
